LIN {X 0,Y 474.663,Z 446.241,A -85,B 0,C 180,E1 -7299.158,E2 -7299.158} C_VEL
LIN {X 0,Y 474.945,Z 438.322,A -85,B 0,C 180,E1 -7299.905,E2 -7299.905} C_VEL
LIN {X 0,Y 475.196,Z 429.952,A -85,B 0,C 180,E1 -7300.546,E2 -7300.546} C_VEL
LIN {X 0,Y 475.533,Z 419.253,A -85,B 0,C 180,E1 -7301.185,E2 -7301.185} C_VEL
LIN {X 0,Y 475.767,Z 407.58,A -85,B 0,C 180,E1 -7301.665,E2 -7301.665} C_VEL
LIN {X 0,Y 476.072,Z 397.775,A -85,B 0,C 180,E1 -7301.927,E2 -7301.927} C_VEL
LIN {X 0,Y 476.288,Z 334.559,A -85,B 0,C 180,E1 -7302.914,E2 -7302.914} C_VEL
LIN {X 0,Y 474.47,Z 320.647,A -85,B 0,C 180,E1 -7303.185,E2 -7303.185} C_VEL
LIN {X 0,Y 474.912,Z 304.767,A -85,B 0,C 180,E1 -7306.33,E2 -7306.33} C_VEL
LIN {X 0,Y 475.219,Z 291.489,A -85,B 0,C 180,E1 -7308.987,E2 -7308.987} C_VEL
LIN {X 0,Y 475.693,Z 278.163,A -85,B 0,C 180,E1 -7311.675,E2 -7311.675} C_VEL
LIN {X 0,Y 474.63,Z 271.177,A -85,B 0,C 180,E1 -7313.207,E2 -7313.207} C_VEL
LIN {X 0,Y 474.589,Z 271.182,A -85,B 0,C 180,E1 -7316.375,E2 -7316.375} C_VEL
LIN {X 0,Y 474.596,Z 271.18,A -85,B 0,C 180,E1 -7319.253,E2 -7319.253} C_VEL
LIN {X 0,Y 474.609,Z 271.177,A -85,B 0,C 180,E1 -7322.429,E2 -7322.429} C_VEL
LIN {X 0,Y 474.607,Z 271.177,A -85,B 0,C 180,E1 -7325.468,E2 -7325.468} C_VEL
LIN {X 0,Y 474.605,Z 271.178,A -85,B 0,C 180,E1 -7328.457,E2 -7328.457} C_VEL
LIN {X 0,Y 474.606,Z 271.176,A -85,B 0,C 180,E1 -7331.785,E2 -7331.785} C_VEL
LIN {X 0,Y 474.608,Z 271.181,A -85,B 0,C 180,E1 -7335.297,E2 -7335.297} C_VEL
LIN {X 0,Y 474.612,Z 271.173,A -85,B 0,C 180,E1 -7338.214,E2 -7338.214} C_VEL
LIN {X 0,Y 474.601,Z 271.181,A -85,B 0,C 180,E1 -7341.542,E2 -7341.542} C_VEL
LIN {X 0,Y 474.617,Z 271.172,A -85,B 0,C 180,E1 -7344.725,E2 -7344.725} C_VEL
LIN {X 0,Y 474.624,Z 271.175,A -85,B 0,C 180,E1 -7347.787,E2 -7347.787} C_VEL
LIN {X 0,Y 474.611,Z 271.172,A -85,B 0,C 180,E1 -7350.884,E2 -7350.884} C_VEL
LIN {X 0,Y 474.641,Z 271.168,A -85,B 0,C 180,E1 -7353.627,E2 -7353.627} C_VEL
LIN {X 0,Y 474.622,Z 271.171,A -85,B 0,C 180,E1 -7356.641,E2 -7356.641} C_VEL
LIN {X 0,Y 474.641,Z 271.173,A -85,B 0,C 180,E1 -7360.089,E2 -7360.089} C_VEL
LIN {X 0,Y 474.633,Z 271.17,A -85,B 0,C 180,E1 -7362.774,E2 -7362.774} C_VEL
LIN {X 0,Y 474.632,Z 271.167,A -85,B 0,C 180,E1 -7365.421,E2 -7365.421} C_VEL
LIN {X 0,Y 474.692,Z 271.165,A -85,B 0,C 180,E1 -7368.037,E2 -7368.037} C_VEL
LIN {X 0,Y 474.714,Z 271.156,A -85,B 0,C 180,E1 -7371.486,E2 -7371.486} C_VEL
LIN {X 0,Y 474.761,Z 271.154,A -85,B 0,C 180,E1 -7374.052,E2 -7374.052} C_VEL
LIN {X 0,Y 474.879,Z 271.138,A -85,B 0,C 180,E1 -7377.455,E2 -7377.455} C_VEL
LIN {X 0,Y 474.844,Z 271.15,A -85,B 0,C 180,E1 -7380.848,E2 -7380.848} C_VEL
LIN {X 0,Y 474.879,Z 271.137,A -85,B 0,C 180,E1 -7382.545,E2 -7382.545} C_VEL
LIN {X 0,Y 474.747,Z 271.155,A -85,B 0,C 180,E1 -7385.948,E2 -7385.948} C_VEL
LIN {X 0,Y 474.714,Z 271.157,A -85,B 0,C 180,E1 -7388.514,E2 -7388.514} C_VEL
LIN {X 0,Y 474.691,Z 271.161,A -85,B 0,C 180,E1 -7391.963,E2 -7391.963} C_VEL
LIN {X 0,Y 474.687,Z 271.172,A -85,B 0,C 180,E1 -7395.456,E2 -7395.456} C_VEL
LIN {X 0,Y 474.652,Z 271.171,A -85,B 0,C 180,E1 -7399.011,E2 -7399.011} C_VEL
LIN {X 0,Y 474.578,Z 271.186,A -85,B 0,C 180,E1 -7401.73,E2 -7401.73} C_VEL
LIN {X 0,Y 474.648,Z 271.171,A -85,B 0,C 180,E1 -7404.494,E2 -7404.494} C_VEL
LIN {X 0,Y 474.689,Z 271.165,A -85,B 0,C 180,E1 -7407.339,E2 -7407.339} C_VEL
LIN {X 0,Y 474.599,Z 271.175,A -85,B 0,C 180,E1 -7410.812,E2 -7410.812} C_VEL
LIN {X 0,Y 474.63,Z 271.178,A -85,B 0,C 180,E1 -7413.985,E2 -7413.985} C_VEL
LIN {X 0,Y 474.567,Z 271.181,A -85,B 0,C 180,E1 -7416.901,E2 -7416.901} C_VEL
LIN {X 0,Y 474.643,Z 271.172,A -85,B 0,C 180,E1 -7419.652,E2 -7419.652} C_VEL
LIN {X 0,Y 474.67,Z 271.173,A -85,B 0,C 180,E1 -7422.928,E2 -7422.928} C_VEL
LIN {X 0,Y 474.739,Z 271.319,A -85,B 0,C 180,E1 -7423.547,E2 -7423.547} C_VEL
LIN {X 0,Y 474.742,Z 280.743,A -85,B 0,C 180,E1 -7425.594,E2 -7425.594} C_VEL
LIN {X 0,Y 474.571,Z 295.866,A -85,B 0,C 180,E1 -7428.877,E2 -7428.877} C_VEL
LIN {X 0,Y 476.56,Z 308.996,A -85,B 0,C 180,E1 -7429.138,E2 -7429.138} C_VEL
LIN {X 0,Y 476.074,Z 372.113,A -85,B 0,C 180,E1 -7430.117,E2 -7430.117} C_VEL
LIN {X 0,Y 475.952,Z 381.875,A -85,B 0,C 180,E1 -7430.383,E2 -7430.383} C_VEL
LIN {X 0,Y 475.739,Z 393.015,A -85,B 0,C 180,E1 -7430.838,E2 -7430.838} C_VEL
LIN {X 0,Y 475.383,Z 404.114,A -85,B 0,C 180,E1 -7431.497,E2 -7431.497} C_VEL
LIN {X 0,Y 475.112,Z 412.388,A -85,B 0,C 180,E1 -7432.131,E2 -7432.131} C_VEL
LIN {X 0,Y 474.847,Z 419.279,A -85,B 0,C 180,E1 -7432.772,E2 -7432.772} C_VEL
LIN {X 0,Y 474.633,Z 425.51,A -85,B 0,C 180,E1 -7433.463,E2 -7433.463} C_VEL
LIN {X 0,Y 474.401,Z 432.473,A -85,B 0,C 180,E1 -7434.401,E2 -7434.401} C_VEL
LIN {X 0,Y 474.202,Z 437.454,A -85,B 0,C 180,E1 -7435.209,E2 -7435.209} C_VEL
LIN {X 0,Y 474.096,Z 442.083,A -85,B 0,C 180,E1 -7436.114,E2 -7436.114} C_VEL
LIN {X 0,Y 473.939,Z 445.242,A -85,B 0,C 180,E1 -7436.845,E2 -7436.845} C_VEL
LIN {X 0,Y 473.214,Z 447.665,A -85,B 0,C 180,E1 -7437.499,E2 -7437.499} C_VEL
LIN {X 0,Y 471.579,Z 449.734,A -85,B 0,C 180,E1 -7438.147,E2 -7438.147} C_VEL
LIN {X 0,Y 467.774,Z 452.844,A -85,B 0,C 180,E1 -7439.474,E2 -7439.474} C_VEL
LIN {X 0,Y 466.671,Z 453.932,A -85,B 0,C 180,E1 -7440.177,E2 -7440.177} C_VEL
LIN {X 0,Y 466.563,Z 454.183,A -85,B 0,C 180,E1 -7440.417,E2 -7440.417} C_VEL
LIN {X 0,Y 466.523,Z 454.848,A -85,B 0,C 180,E1 -7441.18,E2 -7441.18} C_VEL
LIN {X 0,Y 466.5,Z 455.117,A -85,B 0,C 180,E1 -7442.16,E2 -7442.16} C_VEL
LIN {X 0,Y 466.54,Z 454.729,A -85,B 0,C 180,E1 -7443.134,E2 -7443.134} C_VEL
LIN {X 0,Y 466.555,Z 453.682,A -85,B 0,C 180,E1 -7444.098,E2 -7444.098} C_VEL
LIN {X 0,Y 466.732,Z 450.926,A -85,B 0,C 180,E1 -7445.539,E2 -7445.539} C_VEL
LIN {X 0,Y 466.843,Z 447.631,A -85,B 0,C 180,E1 -7446.681,E2 -7446.681} C_VEL
LIN {X 0,Y 466.947,Z 443.943,A -85,B 0,C 180,E1 -7447.665,E2 -7447.665} C_VEL
LIN {X 0,Y 467.086,Z 439.593,A -85,B 0,C 180,E1 -7448.601,E2 -7448.601} C_VEL
LIN {X 0,Y 467.295,Z 434.283,A -85,B 0,C 180,E1 -7449.533,E2 -7449.533} C_VEL
LIN {X 0,Y 467.54,Z 427.826,A -85,B 0,C 180,E1 -7450.461,E2 -7450.461} C_VEL
LIN {X 0,Y 467.766,Z 421.819,A -85,B 0,C 180,E1 -7451.183,E2 -7451.183} C_VEL
LIN {X 0,Y 468.079,Z 413.97,A -85,B 0,C 180,E1 -7451.961,E2 -7451.961} C_VEL
LIN {X 0,Y 468.322,Z 406.975,A -85,B 0,C 180,E1 -7452.535,E2 -7452.535} C_VEL
LIN {X 0,Y 468.602,Z 398.339,A -85,B 0,C 180,E1 -7453.108,E2 -7453.108} C_VEL
LIN {X 0,Y 468.824,Z 390.258,A -85,B 0,C 180,E1 -7453.531,E2 -7453.531} C_VEL
LIN {X 0,Y 468.982,Z 381.301,A -85,B 0,C 180,E1 -7453.885,E2 -7453.885} C_VEL
LIN {X 0,Y 469.169,Z 371.936,A -85,B 0,C 180,E1 -7454.137,E2 -7454.137} C_VEL
LIN {X 0,Y 469.47,Z 308.099,A -85,B 0,C 180,E1 -7455.146,E2 -7455.146} C_VEL
LIN {X 0,Y 467.529,Z 296.318,A -85,B 0,C 180,E1 -7455.389,E2 -7455.389} C_VEL
LIN {X 0,Y 467.842,Z 284.205,A -85,B 0,C 180,E1 -7458.3,E2 -7458.3} C_VEL
LIN {X 0,Y 467.997,Z 275.173,A -85,B 0,C 180,E1 -7460.492,E2 -7460.492} C_VEL
LIN {X 0,Y 467.731,Z 272.039,A -85,B 0,C 180,E1 -7461.304,E2 -7461.304} C_VEL
LIN {X 0,Y 467.736,Z 272.036,A -85,B 0,C 180,E1 -7463.963,E2 -7463.963} C_VEL
LIN {X 0,Y 467.86,Z 272.017,A -85,B 0,C 180,E1 -7467.417,E2 -7467.417} C_VEL
LIN {X 0,Y 467.884,Z 272.018,A -85,B 0,C 180,E1 -7470,E2 -7470} C_VEL
LIN {X 0,Y 467.861,Z 272.015,A -85,B 0,C 180,E1 -7472.583,E2 -7472.583} C_VEL
LIN {X 0,Y 467.722,Z 272.038,A -85,B 0,C 180,E1 -7476.037,E2 -7476.037} C_VEL
LIN {X 0,Y 467.682,Z 272.039,A -85,B 0,C 180,E1 -7478.642,E2 -7478.642} C_VEL
LIN {X 0,Y 467.657,Z 272.045,A -85,B 0,C 180,E1 -7482.145,E2 -7482.145} C_VEL
LIN {X 0,Y 467.64,Z 272.041,A -85,B 0,C 180,E1 -7485.694,E2 -7485.694} C_VEL
LIN {X 0,Y 467.613,Z 272.05,A -85,B 0,C 180,E1 -7488.762,E2 -7488.762} C_VEL
LIN {X 0,Y 467.58,Z 272.05,A -85,B 0,C 180,E1 -7491.267,E2 -7491.267} C_VEL
LIN {X 0,Y 467.57,Z 272.05,A -85,B 0,C 180,E1 -7493.943,E2 -7493.943} C_VEL
LIN {X 0,Y 467.615,Z 272.052,A -85,B 0,C 180,E1 -7496.8,E2 -7496.8} C_VEL
LIN {X 0,Y 467.552,Z 272.052,A -85,B 0,C 180,E1 -7499.737,E2 -7499.737} C_VEL
LIN {X 0,Y 467.576,Z 272.053,A -85,B 0,C 180,E1 -7502.758,E2 -7502.758} C_VEL
LIN {X 0,Y 467.549,Z 272.053,A -85,B 0,C 180,E1 -7505.889,E2 -7505.889} C_VEL
LIN {X 0,Y 467.577,Z 272.055,A -85,B 0,C 180,E1 -7509.144,E2 -7509.144} C_VEL
LIN {X 0,Y 467.581,Z 272.048,A -85,B 0,C 180,E1 -7512.566,E2 -7512.566} C_VEL
LIN {X 0,Y 467.564,Z 272.053,A -85,B 0,C 180,E1 -7515.052,E2 -7515.052} C_VEL
LIN {X 0,Y 467.618,Z 272.05,A -85,B 0,C 180,E1 -7517.443,E2 -7517.443} C_VEL
LIN {X 0,Y 467.592,Z 272.047,A -85,B 0,C 180,E1 -7520.856,E2 -7520.856} C_VEL
LIN {X 0,Y 467.555,Z 272.054,A -85,B 0,C 180,E1 -7524.259,E2 -7524.259} C_VEL
LIN {X 0,Y 467.573,Z 272.05,A -85,B 0,C 180,E1 -7527.32,E2 -7527.32} C_VEL
LIN {X 0,Y 467.568,Z 272.051,A -85,B 0,C 180,E1 -7530.665,E2 -7530.665} C_VEL
LIN {X 0,Y 467.617,Z 272.043,A -85,B 0,C 180,E1 -7533.2,E2 -7533.2} C_VEL
LIN {X 0,Y 467.582,Z 272.054,A -85,B 0,C 180,E1 -7536.467,E2 -7536.467} C_VEL
LIN {X 0,Y 467.611,Z 272.046,A -85,B 0,C 180,E1 -7539.777,E2 -7539.777} C_VEL
LIN {X 0,Y 467.597,Z 272.055,A -85,B 0,C 180,E1 -7542.506,E2 -7542.506} C_VEL
LIN {X 0,Y 467.593,Z 272.048,A -85,B 0,C 180,E1 -7545.196,E2 -7545.196} C_VEL
LIN {X 0,Y 467.643,Z 272.041,A -85,B 0,C 180,E1 -7547.854,E2 -7547.854} C_VEL
LIN {X 0,Y 467.669,Z 272.039,A -85,B 0,C 180,E1 -7551.357,E2 -7551.357} C_VEL
LIN {X 0,Y 467.722,Z 272.03,A -85,B 0,C 180,E1 -7553.962,E2 -7553.962} C_VEL
LIN {X 0,Y 467.846,Z 272.018,A -85,B 0,C 180,E1 -7557.417,E2 -7557.417} C_VEL
LIN {X 0,Y 467.867,Z 272.012,A -85,B 0,C 180,E1 -7560,E2 -7560} C_VEL
LIN {X 0,Y 467.846,Z 272.016,A -85,B 0,C 180,E1 -7562.583,E2 -7562.583} C_VEL
LIN {X 0,Y 467.725,Z 272.031,A -85,B 0,C 180,E1 -7566.038,E2 -7566.038} C_VEL
LIN {X 0,Y 467.669,Z 272.037,A -85,B 0,C 180,E1 -7568.643,E2 -7568.643} C_VEL
LIN {X 0,Y 467.671,Z 272.038,A -85,B 0,C 180,E1 -7572.145,E2 -7572.145} C_VEL
LIN {X 0,Y 467.637,Z 272.047,A -85,B 0,C 180,E1 -7575.885,E2 -7575.885} C_VEL
LIN {X 0,Y 467.611,Z 272.047,A -85,B 0,C 180,E1 -7579.308,E2 -7579.308} C_VEL
LIN {X 0,Y 467.523,Z 272.061,A -85,B 0,C 180,E1 -7582.074,E2 -7582.074} C_VEL
LIN {X 0,Y 467.592,Z 272.047,A -85,B 0,C 180,E1 -7584.888,E2 -7584.888} C_VEL
LIN {X 0,Y 467.608,Z 272.049,A -85,B 0,C 180,E1 -7587.77,E2 -7587.77} C_VEL
LIN {X 0,Y 467.557,Z 272.051,A -85,B 0,C 180,E1 -7591.045,E2 -7591.045} C_VEL
LIN {X 0,Y 467.58,Z 272.056,A -85,B 0,C 180,E1 -7594.243,E2 -7594.243} C_VEL
LIN {X 0,Y 467.539,Z 272.054,A -85,B 0,C 180,E1 -7597.187,E2 -7597.187} C_VEL
LIN {X 0,Y 467.566,Z 272.055,A -85,B 0,C 180,E1 -7600.266,E2 -7600.266} C_VEL
LIN {X 0,Y 467.579,Z 272.057,A -85,B 0,C 180,E1 -7602.568,E2 -7602.568} C_VEL
LIN {X 0,Y 467.558,Z 272.055,A -85,B 0,C 180,E1 -7605.053,E2 -7605.053} C_VEL
LIN {X 0,Y 467.565,Z 272.056,A -85,B 0,C 180,E1 -7608.597,E2 -7608.597} C_VEL
LIN {X 0,Y 467.559,Z 272.051,A -85,B 0,C 180,E1 -7611.956,E2 -7611.956} C_VEL
LIN {X 0,Y 467.553,Z 272.059,A -85,B 0,C 180,E1 -7615.168,E2 -7615.168} C_VEL
LIN {X 0,Y 467.577,Z 272.048,A -85,B 0,C 180,E1 -7618.261,E2 -7618.261} C_VEL
LIN {X 0,Y 467.551,Z 272.061,A -85,B 0,C 180,E1 -7621.25,E2 -7621.25} C_VEL
LIN {X 0,Y 467.565,Z 272.053,A -85,B 0,C 180,E1 -7624.158,E2 -7624.158} C_VEL
LIN {X 0,Y 467.609,Z 272.073,A -85,B 0,C 180,E1 -7626.464,E2 -7626.464} C_VEL
LIN {X 0,Y 468.776,Z 278.945,A -85,B 0,C 180,E1 -7627.988,E2 -7627.988} C_VEL
LIN {X 0,Y 468.56,Z 287.645,A -85,B 0,C 180,E1 -7629.82,E2 -7629.82} C_VEL
LIN {X 0,Y 468.008,Z 303.938,A -85,B 0,C 180,E1 -7633.198,E2 -7633.198} C_VEL
LIN {X 0,Y 467.474,Z 320.66,A -85,B 0,C 180,E1 -7636.619,E2 -7636.619} C_VEL
LIN {X 0,Y 469.474,Z 337.921,A -85,B 0,C 180,E1 -7636.966,E2 -7636.966} C_VEL
LIN {X 0,Y 469.076,Z 398.227,A -85,B 0,C 180,E1 -7637.92,E2 -7637.92} C_VEL
LIN {X 0,Y 468.802,Z 408.676,A -85,B 0,C 180,E1 -7638.214,E2 -7638.214} C_VEL
LIN {X 0,Y 468.482,Z 420.839,A -85,B 0,C 180,E1 -7638.754,E2 -7638.754} C_VEL
LIN {X 0,Y 468.211,Z 429.659,A -85,B 0,C 180,E1 -7639.295,E2 -7639.295} C_VEL
LIN {X 0,Y 467.919,Z 438.06,A -85,B 0,C 180,E1 -7639.945,E2 -7639.945} C_VEL
LIN {X 0,Y 467.619,Z 445.999,A -85,B 0,C 180,E1 -7640.703,E2 -7640.703} C_VEL
LIN {X 0,Y 467.305,Z 453.415,A -85,B 0,C 180,E1 -7641.568,E2 -7641.568} C_VEL
LIN {X 0,Y 467.048,Z 460.937,A -85,B 0,C 180,E1 -7642.652,E2 -7642.652} C_VEL
LIN {X 0,Y 466.87,Z 467.813,A -85,B 0,C 180,E1 -7643.951,E2 -7643.951} C_VEL
LIN {X 0,Y 466.72,Z 473.018,A -85,B 0,C 180,E1 -7645.249,E2 -7645.249} C_VEL
LIN {X 0,Y 466.706,Z 475.684,A -85,B 0,C 180,E1 -7646.115,E2 -7646.115} C_VEL
LIN {X 0,Y 466.666,Z 478.604,A -85,B 0,C 180,E1 -7647.411,E2 -7647.411} C_VEL
LIN {X 0,Y 466.606,Z 479.865,A -85,B 0,C 180,E1 -7648.274,E2 -7648.274} C_VEL
LIN {X 0,Y 466.616,Z 480.652,A -85,B 0,C 180,E1 -7649.137,E2 -7649.137} C_VEL
LIN {X 0,Y 466.597,Z 480.945,A -85,B 0,C 180,E1 -7650,E2 -7650} C_VEL
LIN {X 0,Y 466.616,Z 480.646,A -85,B 0,C 180,E1 -7650.863,E2 -7650.863} C_VEL
LIN {X 0,Y 466.606,Z 479.86,A -85,B 0,C 180,E1 -7651.726,E2 -7651.726} C_VEL
LIN {X 0,Y 466.666,Z 478.599,A -85,B 0,C 180,E1 -7652.589,E2 -7652.589} C_VEL
LIN {X 0,Y 466.706,Z 475.676,A -85,B 0,C 180,E1 -7653.885,E2 -7653.885} C_VEL
LIN {X 0,Y 466.72,Z 473.012,A -85,B 0,C 180,E1 -7654.751,E2 -7654.751} C_VEL
LIN {X 0,Y 466.857,Z 467.805,A -85,B 0,C 180,E1 -7656.049,E2 -7656.049} C_VEL
LIN {X 0,Y 467.048,Z 460.944,A -85,B 0,C 180,E1 -7657.348,E2 -7657.348} C_VEL
LIN {X 0,Y 467.305,Z 453.449,A -85,B 0,C 180,E1 -7658.432,E2 -7658.432} C_VEL
LIN {X 0,Y 467.62,Z 446.06,A -85,B 0,C 180,E1 -7659.297,E2 -7659.297} C_VEL
LIN {X 0,Y 467.938,Z 438.149,A -85,B 0,C 180,E1 -7660.055,E2 -7660.055} C_VEL
LIN {X 0,Y 468.216,Z 429.79,A -85,B 0,C 180,E1 -7660.705,E2 -7660.705} C_VEL
LIN {X 0,Y 468.567,Z 419.109,A -85,B 0,C 180,E1 -7661.353,E2 -7661.353} C_VEL
LIN {X 0,Y 468.837,Z 407.471,A -85,B 0,C 180,E1 -7661.84,E2 -7661.84} C_VEL
LIN {X 0,Y 469.142,Z 397.719,A -85,B 0,C 180,E1 -7662.106,E2 -7662.106} C_VEL
LIN {X 0,Y 469.384,Z 335.49,A -85,B 0,C 180,E1 -7663.093,E2 -7663.093} C_VEL
LIN {X 0,Y 467.442,Z 320.385,A -85,B 0,C 180,E1 -7663.399,E2 -7663.399} C_VEL
LIN {X 0,Y 467.903,Z 304.556,A -85,B 0,C 180,E1 -7666.581,E2 -7666.581} C_VEL
LIN {X 0,Y 468.219,Z 292.753,A -85,B 0,C 180,E1 -7668.98,E2 -7668.98} C_VEL
LIN {X 0,Y 468.703,Z 279.867,A -85,B 0,C 180,E1 -7671.618,E2 -7671.618} C_VEL
LIN {X 0,Y 467.897,Z 273.478,A -85,B 0,C 180,E1 -7672.987,E2 -7672.987} C_VEL
LIN {X 0,Y 467.6,Z 272.053,A -85,B 0,C 180,E1 -7673.315,E2 -7673.315} C_VEL
LIN {X 0,Y 467.564,Z 272.055,A -85,B 0,C 180,E1 -7675.842,E2 -7675.842} C_VEL
LIN {X 0,Y 467.541,Z 272.061,A -85,B 0,C 180,E1 -7678.751,E2 -7678.751} C_VEL
LIN {X 0,Y 467.576,Z 272.05,A -85,B 0,C 180,E1 -7681.739,E2 -7681.739} C_VEL
LIN {X 0,Y 467.553,Z 272.06,A -85,B 0,C 180,E1 -7684.832,E2 -7684.832} C_VEL
LIN {X 0,Y 467.558,Z 272.055,A -85,B 0,C 180,E1 -7688.044,E2 -7688.044} C_VEL
LIN {X 0,Y 467.565,Z 272.057,A -85,B 0,C 180,E1 -7691.403,E2 -7691.403} C_VEL
LIN {X 0,Y 467.558,Z 272.059,A -85,B 0,C 180,E1 -7695.052,E2 -7695.052} C_VEL
LIN {X 0,Y 467.581,Z 272.057,A -85,B 0,C 180,E1 -7697.439,E2 -7697.439} C_VEL
LIN {X 0,Y 467.55,Z 272.054,A -85,B 0,C 180,E1 -7700.852,E2 -7700.852} C_VEL
LIN {X 0,Y 467.552,Z 272.054,A -85,B 0,C 180,E1 -7704.26,E2 -7704.26} C_VEL
LIN {X 0,Y 467.571,Z 272.05,A -85,B 0,C 180,E1 -7707.32,E2 -7707.32} C_VEL
LIN {X 0,Y 467.557,Z 272.051,A -85,B 0,C 180,E1 -7710.667,E2 -7710.667} C_VEL
LIN {X 0,Y 467.601,Z 272.041,A -85,B 0,C 180,E1 -7713.199,E2 -7713.199} C_VEL
LIN {X 0,Y 467.578,Z 272.05,A -85,B 0,C 180,E1 -7716.468,E2 -7716.468} C_VEL
LIN {X 0,Y 467.609,Z 272.044,A -85,B 0,C 180,E1 -7719.777,E2 -7719.777} C_VEL
LIN {X 0,Y 467.592,Z 272.05,A -85,B 0,C 180,E1 -7722.506,E2 -7722.506} C_VEL
LIN {X 0,Y 467.59,Z 272.044,A -85,B 0,C 180,E1 -7725.196,E2 -7725.196} C_VEL
LIN {X 0,Y 467.644,Z 272.042,A -85,B 0,C 180,E1 -7727.854,E2 -7727.854} C_VEL
LIN {X 0,Y 467.668,Z 272.034,A -85,B 0,C 180,E1 -7731.357,E2 -7731.357} C_VEL
LIN {X 0,Y 467.724,Z 272.03,A -85,B 0,C 180,E1 -7733.962,E2 -7733.962} C_VEL
LIN {X 0,Y 467.845,Z 272.014,A -85,B 0,C 180,E1 -7737.417,E2 -7737.417} C_VEL
LIN {X 0,Y 467.866,Z 272.012,A -85,B 0,C 180,E1 -7740,E2 -7740} C_VEL
LIN {X 0,Y 467.845,Z 272.013,A -85,B 0,C 180,E1 -7742.583,E2 -7742.583} C_VEL
LIN {X 0,Y 467.709,Z 272.032,A -85,B 0,C 180,E1 -7746.038,E2 -7746.038} C_VEL
LIN {X 0,Y 467.668,Z 272.036,A -85,B 0,C 180,E1 -7748.643,E2 -7748.643} C_VEL
LIN {X 0,Y 467.643,Z 272.037,A -85,B 0,C 180,E1 -7752.146,E2 -7752.146} C_VEL
LIN {X 0,Y 467.626,Z 272.047,A -85,B 0,C 180,E1 -7755.696,E2 -7755.696} C_VEL
LIN {X 0,Y 467.605,Z 272.048,A -85,B 0,C 180,E1 -7758.765,E2 -7758.765} C_VEL
LIN {X 0,Y 467.569,Z 272.053,A -85,B 0,C 180,E1 -7761.269,E2 -7761.269} C_VEL
LIN {X 0,Y 467.562,Z 272.058,A -85,B 0,C 180,E1 -7763.944,E2 -7763.944} C_VEL
LIN {X 0,Y 467.617,Z 272.044,A -85,B 0,C 180,E1 -7766.8,E2 -7766.8} C_VEL
LIN {X 0,Y 467.576,Z 272.054,A -85,B 0,C 180,E1 -7769.737,E2 -7769.737} C_VEL
LIN {X 0,Y 467.574,Z 272.052,A -85,B 0,C 180,E1 -7772.759,E2 -7772.759} C_VEL
LIN {X 0,Y 467.548,Z 272.056,A -85,B 0,C 180,E1 -7775.89,E2 -7775.89} C_VEL
LIN {X 0,Y 467.592,Z 272.05,A -85,B 0,C 180,E1 -7779.144,E2 -7779.144} C_VEL
LIN {X 0,Y 467.613,Z 272.053,A -85,B 0,C 180,E1 -7782.572,E2 -7782.572} C_VEL
LIN {X 0,Y 467.692,Z 272.169,A -85,B 0,C 180,E1 -7783.431,E2 -7783.431} C_VEL
LIN {X 0,Y 467.757,Z 280.981,A -85,B 0,C 180,E1 -7785.372,E2 -7785.372} C_VEL
LIN {X 0,Y 467.529,Z 295.966,A -85,B 0,C 180,E1 -7788.662,E2 -7788.662} C_VEL
LIN {X 0,Y 469.614,Z 308.501,A -85,B 0,C 180,E1 -7788.928,E2 -7788.928} C_VEL
LIN {X 0,Y 469.139,Z 372.245,A -85,B 0,C 180,E1 -7789.933,E2 -7789.933} C_VEL
LIN {X 0,Y 469.024,Z 381.964,A -85,B 0,C 180,E1 -7790.201,E2 -7790.201} C_VEL
LIN {X 0,Y 468.818,Z 392.478,A -85,B 0,C 180,E1 -7790.633,E2 -7790.633} C_VEL
LIN {X 0,Y 468.438,Z 403.494,A -85,B 0,C 180,E1 -7791.275,E2 -7791.275} C_VEL
LIN {X 0,Y 468.105,Z 412.934,A -85,B 0,C 180,E1 -7792.009,E2 -7792.009} C_VEL
LIN {X 0,Y 467.803,Z 420.829,A -85,B 0,C 180,E1 -7792.773,E2 -7792.773} C_VEL
LIN {X 0,Y 467.546,Z 427.649,A -85,B 0,C 180,E1 -7793.578,E2 -7793.578} C_VEL
LIN {X 0,Y 467.287,Z 434.861,A -85,B 0,C 180,E1 -7794.618,E2 -7794.618} C_VEL
LIN {X 0,Y 467.046,Z 441.555,A -85,B 0,C 180,E1 -7795.856,E2 -7795.856} C_VEL
LIN {X 0,Y 466.865,Z 445.626,A -85,B 0,C 180,E1 -7796.813,E2 -7796.813} C_VEL
LIN {X 0,Y 466.76,Z 450.059,A -85,B 0,C 180,E1 -7798.199,E2 -7798.199} C_VEL
LIN {X 0,Y 466.667,Z 452.364,A -85,B 0,C 180,E1 -7799.201,E2 -7799.201} C_VEL
LIN {X 0,Y 466.563,Z 454.183,A -85,B 0,C 180,E1 -7800.417,E2 -7800.417} C_VEL
LIN {X 0,Y 465.835,Z 454.858,A -85,B 0,C 180,E1 -7801.133,E2 -7801.133} C_VEL
LIN {X 0,Y 462.926,Z 455.162,A -85,B 0,C 180,E1 -7802.302,E2 -7802.302} C_VEL
LIN {X 0,Y 460.075,Z 454.587,A -85,B 0,C 180,E1 -7803.484,E2 -7803.484} C_VEL
LIN {X 0,Y 459.453,Z 453.679,A -85,B 0,C 180,E1 -7804.213,E2 -7804.213} C_VEL
LIN {X 0,Y 459.653,Z 451.038,A -85,B 0,C 180,E1 -7805.618,E2 -7805.618} C_VEL
LIN {X 0,Y 459.744,Z 448.396,A -85,B 0,C 180,E1 -7806.582,E2 -7806.582} C_VEL
LIN {X 0,Y 459.878,Z 444.004,A -85,B 0,C 180,E1 -7807.776,E2 -7807.776} C_VEL
LIN {X 0,Y 460.026,Z 439.568,A -85,B 0,C 180,E1 -7808.737,E2 -7808.737} C_VEL
LIN {X 0,Y 460.25,Z 434.28,A -85,B 0,C 180,E1 -7809.673,E2 -7809.673} C_VEL
LIN {X 0,Y 460.521,Z 428.073,A -85,B 0,C 180,E1 -7810.577,E2 -7810.577} C_VEL
LIN {X 0,Y 460.798,Z 420.905,A -85,B 0,C 180,E1 -7811.436,E2 -7811.436} C_VEL
LIN {X 0,Y 461.111,Z 413.802,A -85,B 0,C 180,E1 -7812.138,E2 -7812.138} C_VEL
LIN {X 0,Y 461.371,Z 406.725,A -85,B 0,C 180,E1 -7812.721,E2 -7812.721} C_VEL
LIN {X 0,Y 461.634,Z 398.122,A -85,B 0,C 180,E1 -7813.294,E2 -7813.294} C_VEL
LIN {X 0,Y 461.867,Z 390.139,A -85,B 0,C 180,E1 -7813.713,E2 -7813.713} C_VEL
LIN {X 0,Y 462.045,Z 380.541,A -85,B 0,C 180,E1 -7814.091,E2 -7814.091} C_VEL
LIN {X 0,Y 462.232,Z 370.811,A -85,B 0,C 180,E1 -7814.343,E2 -7814.343} C_VEL
LIN {X 0,Y 462.478,Z 308.494,A -85,B 0,C 180,E1 -7815.339,E2 -7815.339} C_VEL
LIN {X 0,Y 460.484,Z 296.423,A -85,B 0,C 180,E1 -7815.612,E2 -7815.612} C_VEL
LIN {X 0,Y 460.831,Z 284.28,A -85,B 0,C 180,E1 -7818.565,E2 -7818.565} C_VEL
LIN {X 0,Y 460.928,Z 275.249,A -85,B 0,C 180,E1 -7820.788,E2 -7820.788} C_VEL
LIN {X 0,Y 460.722,Z 272.912,A -85,B 0,C 180,E1 -7821.392,E2 -7821.392} C_VEL
LIN {X 0,Y 460.695,Z 272.906,A -85,B 0,C 180,E1 -7824.748,E2 -7824.748} C_VEL
LIN {X 0,Y 460.801,Z 272.895,A -85,B 0,C 180,E1 -7827.378,E2 -7827.378} C_VEL
LIN {X 0,Y 460.855,Z 272.894,A -85,B 0,C 180,E1 -7830,E2 -7830} C_VEL
LIN {X 0,Y 460.802,Z 272.894,A -85,B 0,C 180,E1 -7832.622,E2 -7832.622} C_VEL
LIN {X 0,Y 460.686,Z 272.916,A -85,B 0,C 180,E1 -7836.13,E2 -7836.13} C_VEL
LIN {X 0,Y 460.629,Z 272.916,A -85,B 0,C 180,E1 -7838.776,E2 -7838.776} C_VEL
LIN {X 0,Y 460.615,Z 272.924,A -85,B 0,C 180,E1 -7842.444,E2 -7842.444} C_VEL
LIN {X 0,Y 460.601,Z 272.92,A -85,B 0,C 180,E1 -7845.997,E2 -7845.997} C_VEL
LIN {X 0,Y 460.568,Z 272.922,A -85,B 0,C 180,E1 -7849.615,E2 -7849.615} C_VEL
LIN {X 0,Y 460.511,Z 272.934,A -85,B 0,C 180,E1 -7852.428,E2 -7852.428} C_VEL
LIN {X 0,Y 460.556,Z 272.923,A -85,B 0,C 180,E1 -7855.798,E2 -7855.798} C_VEL
LIN {X 0,Y 460.551,Z 272.925,A -85,B 0,C 180,E1 -7858.232,E2 -7858.232} C_VEL
LIN {X 0,Y 460.518,Z 272.933,A -85,B 0,C 180,E1 -7861.282,E2 -7861.282} C_VEL
LIN {X 0,Y 460.519,Z 272.929,A -85,B 0,C 180,E1 -7864.503,E2 -7864.503} C_VEL
LIN {X 0,Y 460.497,Z 272.934,A -85,B 0,C 180,E1 -7867.622,E2 -7867.622} C_VEL
LIN {X 0,Y 460.537,Z 272.926,A -85,B 0,C 180,E1 -7870.268,E2 -7870.268} C_VEL
LIN {X 0,Y 460.495,Z 272.939,A -85,B 0,C 180,E1 -7873.374,E2 -7873.374} C_VEL
LIN {X 0,Y 460.518,Z 272.928,A -85,B 0,C 180,E1 -7876.627,E2 -7876.627} C_VEL
LIN {X 0,Y 460.552,Z 272.932,A -85,B 0,C 180,E1 -7879.727,E2 -7879.727} C_VEL
LIN {X 0,Y 460.52,Z 272.928,A -85,B 0,C 180,E1 -7882.518,E2 -7882.518} C_VEL
LIN {X 0,Y 460.54,Z 272.93,A -85,B 0,C 180,E1 -7885.623,E2 -7885.623} C_VEL
LIN {X 0,Y 460.528,Z 272.927,A -85,B 0,C 180,E1 -7888.744,E2 -7888.744} C_VEL
LIN {X 0,Y 460.549,Z 272.928,A -85,B 0,C 180,E1 -7891.767,E2 -7891.767} C_VEL
LIN {X 0,Y 460.549,Z 272.926,A -85,B 0,C 180,E1 -7894.705,E2 -7894.705} C_VEL
LIN {X 0,Y 460.5,Z 272.931,A -85,B 0,C 180,E1 -7897.571,E2 -7897.571} C_VEL
LIN {X 0,Y 460.557,Z 272.932,A -85,B 0,C 180,E1 -7900.384,E2 -7900.384} C_VEL
LIN {X 0,Y 460.553,Z 272.925,A -85,B 0,C 180,E1 -7903.146,E2 -7903.146} C_VEL
LIN {X 0,Y 460.545,Z 272.925,A -85,B 0,C 180,E1 -7905.868,E2 -7905.868} C_VEL
LIN {X 0,Y 460.598,Z 272.925,A -85,B 0,C 180,E1 -7908.559,E2 -7908.559} C_VEL
LIN {X 0,Y 460.682,Z 272.908,A -85,B 0,C 180,E1 -7912.108,E2 -7912.108} C_VEL
LIN {X 0,Y 460.681,Z 272.914,A -85,B 0,C 180,E1 -7914.748,E2 -7914.748} C_VEL
LIN {X 0,Y 460.811,Z 272.895,A -85,B 0,C 180,E1 -7917.377,E2 -7917.377} C_VEL
LIN {X 0,Y 460.838,Z 272.888,A -85,B 0,C 180,E1 -7920,E2 -7920} C_VEL
LIN {X 0,Y 460.787,Z 272.896,A -85,B 0,C 180,E1 -7922.622,E2 -7922.622} C_VEL
LIN {X 0,Y 460.691,Z 272.907,A -85,B 0,C 180,E1 -7926.13,E2 -7926.13} C_VEL
LIN {X 0,Y 460.616,Z 272.917,A -85,B 0,C 180,E1 -7928.776,E2 -7928.776} C_VEL
LIN {X 0,Y 460.622,Z 272.915,A -85,B 0,C 180,E1 -7932.457,E2 -7932.457} C_VEL
LIN {X 0,Y 460.588,Z 272.923,A -85,B 0,C 180,E1 -7935.998,E2 -7935.998} C_VEL
LIN {X 0,Y 460.558,Z 272.923,A -85,B 0,C 180,E1 -7938.902,E2 -7938.902} C_VEL
LIN {X 0,Y 460.504,Z 272.933,A -85,B 0,C 180,E1 -7941.486,E2 -7941.486} C_VEL
LIN {X 0,Y 460.531,Z 272.93,A -85,B 0,C 180,E1 -7944.333,E2 -7944.333} C_VEL
LIN {X 0,Y 460.561,Z 272.923,A -85,B 0,C 180,E1 -7947.244,E2 -7947.244} C_VEL
LIN {X 0,Y 460.499,Z 272.938,A -85,B 0,C 180,E1 -7950.241,E2 -7950.241} C_VEL
LIN {X 0,Y 460.519,Z 272.928,A -85,B 0,C 180,E1 -7953.326,E2 -7953.326} C_VEL
LIN {X 0,Y 460.468,Z 272.941,A -85,B 0,C 180,E1 -7956.53,E2 -7956.53} C_VEL
LIN {X 0,Y 460.516,Z 272.929,A -85,B 0,C 180,E1 -7959.864,E2 -7959.864} C_VEL
LIN {X 0,Y 460.505,Z 272.934,A -85,B 0,C 180,E1 -7962.901,E2 -7962.901} C_VEL
LIN {X 0,Y 460.498,Z 272.93,A -85,B 0,C 180,E1 -7965.832,E2 -7965.832} C_VEL
LIN {X 0,Y 460.52,Z 272.934,A -85,B 0,C 180,E1 -7968.989,E2 -7968.989} C_VEL
LIN {X 0,Y 460.515,Z 272.932,A -85,B 0,C 180,E1 -7971.267,E2 -7971.267} C_VEL
LIN {X 0,Y 460.503,Z 272.932,A -85,B 0,C 180,E1 -7974.555,E2 -7974.555} C_VEL
LIN {X 0,Y 460.525,Z 272.929,A -85,B 0,C 180,E1 -7977.716,E2 -7977.716} C_VEL
LIN {X 0,Y 460.522,Z 272.93,A -85,B 0,C 180,E1 -7980.769,E2 -7980.769} C_VEL
LIN {X 0,Y 460.516,Z 272.934,A -85,B 0,C 180,E1 -7983.733,E2 -7983.733} C_VEL
LIN {X 0,Y 460.581,Z 273.028,A -85,B 0,C 180,E1 -7986.336,E2 -7986.336} C_VEL
LIN {X 0,Y 461.848,Z 281.163,A -85,B 0,C 180,E1 -7988.162,E2 -7988.162} C_VEL
LIN {X 0,Y 461.425,Z 291.788,A -85,B 0,C 180,E1 -7990.423,E2 -7990.423} C_VEL
LIN {X 0,Y 460.838,Z 308.349,A -85,B 0,C 180,E1 -7993.9,E2 -7993.9} C_VEL
LIN {X 0,Y 460.416,Z 320.573,A -85,B 0,C 180,E1 -7996.435,E2 -7996.435} C_VEL
LIN {X 0,Y 462.542,Z 337.9,A -85,B 0,C 180,E1 -7996.776,E2 -7996.776} C_VEL
LIN {X 0,Y 462.148,Z 397.722,A -85,B 0,C 180,E1 -7997.736,E2 -7997.736} C_VEL
LIN {X 0,Y 461.878,Z 407.449,A -85,B 0,C 180,E1 -7998.007,E2 -7998.007} C_VEL
LIN {X 0,Y 461.609,Z 418.533,A -85,B 0,C 180,E1 -7998.473,E2 -7998.473} C_VEL
LIN {X 0,Y 461.207,Z 429.372,A -85,B 0,C 180,E1 -7999.131,E2 -7999.131} C_VEL
LIN {X 0,Y 460.919,Z 437.791,A -85,B 0,C 180,E1 -7999.79,E2 -7999.79} C_VEL
LIN {X 0,Y 460.575,Z 445.742,A -85,B 0,C 180,E1 -8000.559,E2 -8000.559} C_VEL
LIN {X 0,Y 460.259,Z 453.168,A -85,B 0,C 180,E1 -8001.438,E2 -8001.438} C_VEL
LIN {X 0,Y 459.977,Z 460.701,A -85,B 0,C 180,E1 -8002.538,E2 -8002.538} C_VEL
LIN {X 0,Y 459.781,Z 467.592,A -85,B 0,C 180,E1 -8003.858,E2 -8003.858} C_VEL
LIN {X 0,Y 459.651,Z 472.804,A -85,B 0,C 180,E1 -8005.176,E2 -8005.176} C_VEL
LIN {X 0,Y 459.6,Z 475.475,A -85,B 0,C 180,E1 -8006.054,E2 -8006.054} C_VEL
LIN {X 0,Y 459.59,Z 478.4,A -85,B 0,C 180,E1 -8007.371,E2 -8007.371} C_VEL
LIN {X 0,Y 459.519,Z 479.665,A -85,B 0,C 180,E1 -8008.247,E2 -8008.247} C_VEL
LIN {X 0,Y 459.519,Z 480.454,A -85,B 0,C 180,E1 -8009.124,E2 -8009.124} C_VEL
LIN {X 0,Y 459.529,Z 480.749,A -85,B 0,C 180,E1 -8010,E2 -8010} C_VEL
LIN {X 0,Y 459.519,Z 480.451,A -85,B 0,C 180,E1 -8010.876,E2 -8010.876} C_VEL
LIN {X 0,Y 459.519,Z 479.667,A -85,B 0,C 180,E1 -8011.753,E2 -8011.753} C_VEL
LIN {X 0,Y 459.59,Z 478.409,A -85,B 0,C 180,E1 -8012.629,E2 -8012.629} C_VEL
LIN {X 0,Y 459.6,Z 475.487,A -85,B 0,C 180,E1 -8013.946,E2 -8013.946} C_VEL
LIN {X 0,Y 459.651,Z 472.828,A -85,B 0,C 180,E1 -8014.824,E2 -8014.824} C_VEL
LIN {X 0,Y 459.769,Z 467.621,A -85,B 0,C 180,E1 -8016.142,E2 -8016.142} C_VEL
LIN {X 0,Y 459.977,Z 460.765,A -85,B 0,C 180,E1 -8017.462,E2 -8017.462} C_VEL
LIN {X 0,Y 460.259,Z 453.273,A -85,B 0,C 180,E1 -8018.562,E2 -8018.562} C_VEL
LIN {X 0,Y 460.584,Z 445.888,A -85,B 0,C 180,E1 -8019.441,E2 -8019.441} C_VEL
LIN {X 0,Y 460.923,Z 437.981,A -85,B 0,C 180,E1 -8020.21,E2 -8020.21} C_VEL
LIN {X 0,Y 461.242,Z 429.629,A -85,B 0,C 180,E1 -8020.868,E2 -8020.868} C_VEL
LIN {X 0,Y 461.617,Z 418.965,A -85,B 0,C 180,E1 -8021.526,E2 -8021.526} C_VEL
LIN {X 0,Y 461.901,Z 407.361,A -85,B 0,C 180,E1 -8022.02,E2 -8022.02} C_VEL
LIN {X 0,Y 462.225,Z 397.665,A -85,B 0,C 180,E1 -8022.29,E2 -8022.29} C_VEL
LIN {X 0,Y 462.533,Z 336.585,A -85,B 0,C 180,E1 -8023.275,E2 -8023.275} C_VEL
LIN {X 0,Y 460.399,Z 320.128,A -85,B 0,C 180,E1 -8023.624,E2 -8023.624} C_VEL
LIN {X 0,Y 460.864,Z 305.592,A -85,B 0,C 180,E1 -8026.591,E2 -8026.591} C_VEL
LIN {X 0,Y 461.417,Z 289.981,A -85,B 0,C 180,E1 -8029.809,E2 -8029.809} C_VEL
LIN {X 0,Y 461.658,Z 279.406,A -85,B 0,C 180,E1 -8032.019,E2 -8032.019} C_VEL
LIN {X 0,Y 460.558,Z 272.93,A -85,B 0,C 180,E1 -8033.491,E2 -8033.491} C_VEL
LIN {X 0,Y 460.516,Z 272.935,A -85,B 0,C 180,E1 -8036.267,E2 -8036.267} C_VEL
LIN {X 0,Y 460.516,Z 272.934,A -85,B 0,C 180,E1 -8039.232,E2 -8039.232} C_VEL
LIN {X 0,Y 460.525,Z 272.93,A -85,B 0,C 180,E1 -8042.284,E2 -8042.284} C_VEL
LIN {X 0,Y 460.503,Z 272.935,A -85,B 0,C 180,E1 -8045.445,E2 -8045.445} C_VEL
LIN {X 0,Y 460.532,Z 272.936,A -85,B 0,C 180,E1 -8048.896,E2 -8048.896} C_VEL
LIN {X 0,Y 460.496,Z 272.932,A -85,B 0,C 180,E1 -8052.183,E2 -8052.183} C_VEL
LIN {X 0,Y 460.506,Z 272.937,A -85,B 0,C 180,E1 -8055.41,E2 -8055.41} C_VEL
LIN {X 0,Y 460.523,Z 272.927,A -85,B 0,C 180,E1 -8058.397,E2 -8058.397} C_VEL
LIN {X 0,Y 460.509,Z 272.935,A -85,B 0,C 180,E1 -8061.265,E2 -8061.265} C_VEL
LIN {X 0,Y 460.502,Z 272.931,A -85,B 0,C 180,E1 -8064.554,E2 -8064.554} C_VEL
LIN {X 0,Y 460.52,Z 272.931,A -85,B 0,C 180,E1 -8067.715,E2 -8067.715} C_VEL
LIN {X 0,Y 460.527,Z 272.927,A -85,B 0,C 180,E1 -8070.768,E2 -8070.768} C_VEL
LIN {X 0,Y 460.544,Z 272.925,A -85,B 0,C 180,E1 -8073.734,E2 -8073.734} C_VEL
LIN {X 0,Y 460.532,Z 272.926,A -85,B 0,C 180,E1 -8076.623,E2 -8076.623} C_VEL
LIN {X 0,Y 460.538,Z 272.923,A -85,B 0,C 180,E1 -8079.452,E2 -8079.452} C_VEL
LIN {X 0,Y 460.544,Z 272.933,A -85,B 0,C 180,E1 -8082.23,E2 -8082.23} C_VEL
LIN {X 0,Y 460.55,Z 272.922,A -85,B 0,C 180,E1 -8084.964,E2 -8084.964} C_VEL
LIN {X 0,Y 460.6,Z 272.924,A -85,B 0,C 180,E1 -8088.559,E2 -8088.559} C_VEL
LIN {X 0,Y 460.682,Z 272.906,A -85,B 0,C 180,E1 -8092.108,E2 -8092.108} C_VEL
LIN {X 0,Y 460.683,Z 272.913,A -85,B 0,C 180,E1 -8094.748,E2 -8094.748} C_VEL
LIN {X 0,Y 460.786,Z 272.894,A -85,B 0,C 180,E1 -8097.378,E2 -8097.378} C_VEL
LIN {X 0,Y 460.837,Z 272.888,A -85,B 0,C 180,E1 -8100,E2 -8100} C_VEL
LIN {X 0,Y 460.786,Z 272.893,A -85,B 0,C 180,E1 -8102.623,E2 -8102.623} C_VEL
LIN {X 0,Y 460.673,Z 272.908,A -85,B 0,C 180,E1 -8106.131,E2 -8106.131} C_VEL
LIN {X 0,Y 460.615,Z 272.915,A -85,B 0,C 180,E1 -8108.776,E2 -8108.776} C_VEL
LIN {X 0,Y 460.596,Z 272.915,A -85,B 0,C 180,E1 -8112.335,E2 -8112.335} C_VEL
LIN {X 0,Y 460.588,Z 272.92,A -85,B 0,C 180,E1 -8115.998,E2 -8115.998} C_VEL
LIN {X 0,Y 460.558,Z 272.926,A -85,B 0,C 180,E1 -8118.902,E2 -8118.902} C_VEL
LIN {X 0,Y 460.504,Z 272.935,A -85,B 0,C 180,E1 -8121.486,E2 -8121.486} C_VEL
LIN {X 0,Y 460.532,Z 272.931,A -85,B 0,C 180,E1 -8124.333,E2 -8124.333} C_VEL
LIN {X 0,Y 460.574,Z 272.922,A -85,B 0,C 180,E1 -8127.244,E2 -8127.244} C_VEL
LIN {X 0,Y 460.516,Z 272.934,A -85,B 0,C 180,E1 -8130.24,E2 -8130.24} C_VEL
LIN {X 0,Y 460.52,Z 272.93,A -85,B 0,C 180,E1 -8133.326,E2 -8133.326} C_VEL
LIN {X 0,Y 460.471,Z 272.941,A -85,B 0,C 180,E1 -8136.53,E2 -8136.53} C_VEL
LIN {X 0,Y 460.567,Z 272.927,A -85,B 0,C 180,E1 -8139.859,E2 -8139.859} C_VEL
LIN {X 0,Y 460.616,Z 272.933,A -85,B 0,C 180,E1 -8143.289,E2 -8143.289} C_VEL
LIN {X 0,Y 460.841,Z 277.032,A -85,B 0,C 180,E1 -8144.214,E2 -8144.214} C_VEL
LIN {X 0,Y 460.595,Z 291.658,A -85,B 0,C 180,E1 -8147.457,E2 -8147.457} C_VEL
LIN {X 0,Y 460.518,Z 296.102,A -85,B 0,C 180,E1 -8148.441,E2 -8148.441} C_VEL
LIN {X 0,Y 462.757,Z 309.678,A -85,B 0,C 180,E1 -8148.742,E2 -8148.742} C_VEL
LIN {X 0,Y 462.218,Z 373.22,A -85,B 0,C 180,E1 -8149.763,E2 -8149.763} C_VEL
LIN {X 0,Y 462.035,Z 384.102,A -85,B 0,C 180,E1 -8150.082,E2 -8150.082} C_VEL
LIN {X 0,Y 461.84,Z 394.801,A -85,B 0,C 180,E1 -8150.565,E2 -8150.565} C_VEL
LIN {X 0,Y 461.476,Z 404.167,A -85,B 0,C 180,E1 -8151.143,E2 -8151.143} C_VEL
LIN {X 0,Y 461.12,Z 413.495,A -85,B 0,C 180,E1 -8151.885,E2 -8151.885} C_VEL
LIN {X 0,Y 460.843,Z 420.193,A -85,B 0,C 180,E1 -8152.538,E2 -8152.538} C_VEL
LIN {X 0,Y 460.539,Z 427.058,A -85,B 0,C 180,E1 -8153.342,E2 -8153.342} C_VEL
LIN {X 0,Y 460.358,Z 431.91,A -85,B 0,C 180,E1 -8154.01,E2 -8154.01} C_VEL
LIN {X 0,Y 460.084,Z 438.176,A -85,B 0,C 180,E1 -8155.053,E2 -8155.053} C_VEL
LIN {X 0,Y 459.951,Z 443.274,A -85,B 0,C 180,E1 -8156.108,E2 -8156.108} C_VEL
LIN {X 0,Y 459.787,Z 446.62,A -85,B 0,C 180,E1 -8156.954,E2 -8156.954} C_VEL
LIN {X 0,Y 459.745,Z 448.987,A -85,B 0,C 180,E1 -8157.655,E2 -8157.655} C_VEL
LIN {X 0,Y 459.64,Z 452.093,A -85,B 0,C 180,E1 -8158.899,E2 -8158.899} C_VEL
LIN {X 0,Y 459.523,Z 453.544,A -85,B 0,C 180,E1 -8159.689,E2 -8159.689} C_VEL
LIN {X 0,Y 459.442,Z 454.719,A -85,B 0,C 180,E1 -8160.693,E2 -8160.693} C_VEL
LIN {X 0,Y 459.415,Z 455.235,A -85,B 0,C 180,E1 -8161.692,E2 -8161.692} C_VEL
LIN {X 0,Y 459.427,Z 455.117,A -85,B 0,C 180,E1 -8162.684,E2 -8162.684} C_VEL
LIN {X 0,Y 459.453,Z 453.679,A -85,B 0,C 180,E1 -8164.213,E2 -8164.213} C_VEL
LIN {X 0,Y 458.849,Z 452.589,A -85,B 0,C 180,E1 -8164.935,E2 -8164.935} C_VEL
LIN {X 0,Y 456.12,Z 450.122,A -85,B 0,C 180,E1 -8166.09,E2 -8166.09} C_VEL
LIN {X 0,Y 453.822,Z 447.462,A -85,B 0,C 180,E1 -8166.993,E2 -8166.993} C_VEL
LIN {X 0,Y 452.872,Z 445.018,A -85,B 0,C 180,E1 -8167.667,E2 -8167.667} C_VEL
LIN {X 0,Y 452.816,Z 444.074,A -85,B 0,C 180,E1 -8167.889,E2 -8167.889} C_VEL
LIN {X 0,Y 452.962,Z 439.722,A -85,B 0,C 180,E1 -8168.843,E2 -8168.843} C_VEL
LIN {X 0,Y 453.215,Z 434.273,A -85,B 0,C 180,E1 -8169.817,E2 -8169.817} C_VEL
LIN {X 0,Y 453.514,Z 427.545,A -85,B 0,C 180,E1 -8170.798,E2 -8170.798} C_VEL
LIN {X 0,Y 453.803,Z 420.806,A -85,B 0,C 180,E1 -8171.607,E2 -8171.607} C_VEL
LIN {X 0,Y 454.118,Z 413.654,A -85,B 0,C 180,E1 -8172.319,E2 -8172.319} C_VEL
LIN {X 0,Y 454.476,Z 405.433,A -85,B 0,C 180,E1 -8172.989,E2 -8172.989} C_VEL
LIN {X 0,Y 454.764,Z 395.9,A -85,B 0,C 180,E1 -8173.605,E2 -8173.605} C_VEL
LIN {X 0,Y 455.046,Z 383.555,A -85,B 0,C 180,E1 -8174.176,E2 -8174.176} C_VEL
LIN {X 0,Y 455.301,Z 373.496,A -85,B 0,C 180,E1 -8174.472,E2 -8174.472} C_VEL
LIN {X 0,Y 455.546,Z 338.738,A -85,B 0,C 180,E1 -8175.053,E2 -8175.053} C_VEL
LIN {X 0,Y 455.672,Z 309.961,A -85,B 0,C 180,E1 -8175.514,E2 -8175.514} C_VEL
LIN {X 0,Y 453.482,Z 296.603,A -85,B 0,C 180,E1 -8175.815,E2 -8175.815} C_VEL
LIN {X 0,Y 453.829,Z 284.331,A -85,B 0,C 180,E1 -8178.839,E2 -8178.839} C_VEL
LIN {X 0,Y 453.956,Z 277.083,A -85,B 0,C 180,E1 -8180.645,E2 -8180.645} C_VEL
LIN {X 0,Y 453.672,Z 273.79,A -85,B 0,C 180,E1 -8181.537,E2 -8181.537} C_VEL
LIN {X 0,Y 453.668,Z 273.781,A -85,B 0,C 180,E1 -8184.667,E2 -8184.667} C_VEL
LIN {X 0,Y 453.745,Z 273.774,A -85,B 0,C 180,E1 -8187.337,E2 -8187.337} C_VEL
LIN {X 0,Y 453.825,Z 273.769,A -85,B 0,C 180,E1 -8190,E2 -8190} C_VEL
LIN {X 0,Y 453.746,Z 273.773,A -85,B 0,C 180,E1 -8192.663,E2 -8192.663} C_VEL
LIN {X 0,Y 453.652,Z 273.791,A -85,B 0,C 180,E1 -8196.225,E2 -8196.225} C_VEL
LIN {X 0,Y 453.592,Z 273.792,A -85,B 0,C 180,E1 -8198.913,E2 -8198.913} C_VEL
LIN {X 0,Y 453.565,Z 273.8,A -85,B 0,C 180,E1 -8202.528,E2 -8202.528} C_VEL
LIN {X 0,Y 453.545,Z 273.801,A -85,B 0,C 180,E1 -8206.195,E2 -8206.195} C_VEL
LIN {X 0,Y 453.517,Z 273.803,A -85,B 0,C 180,E1 -8209.039,E2 -8209.039} C_VEL
LIN {X 0,Y 453.476,Z 273.805,A -85,B 0,C 180,E1 -8211.835,E2 -8211.835} C_VEL
LIN {X 0,Y 453.506,Z 273.81,A -85,B 0,C 180,E1 -8214.734,E2 -8214.734} C_VEL
LIN {X 0,Y 453.531,Z 273.798,A -85,B 0,C 180,E1 -8217.959,E2 -8217.959} C_VEL
LIN {X 0,Y 453.462,Z 273.809,A -85,B 0,C 180,E1 -8221.524,E2 -8221.524} C_VEL
LIN {X 0,Y 453.479,Z 273.808,A -85,B 0,C 180,E1 -8224.775,E2 -8224.775} C_VEL
LIN {X 0,Y 453.46,Z 273.807,A -85,B 0,C 180,E1 -8228.311,E2 -8228.311} C_VEL
LIN {X 0,Y 453.489,Z 273.804,A -85,B 0,C 180,E1 -8230.608,E2 -8230.608} C_VEL
LIN {X 0,Y 453.451,Z 273.814,A -85,B 0,C 180,E1 -8233.243,E2 -8233.243} C_VEL
LIN {X 0,Y 453.471,Z 273.811,A -85,B 0,C 180,E1 -8235.779,E2 -8235.779} C_VEL
LIN {X 0,Y 453.49,Z 273.805,A -85,B 0,C 180,E1 -8238.21,E2 -8238.21} C_VEL
LIN {X 0,Y 453.519,Z 273.8,A -85,B 0,C 180,E1 -8240.787,E2 -8240.787} C_VEL
LIN {X 0,Y 453.449,Z 273.816,A -85,B 0,C 180,E1 -8243.917,E2 -8243.917} C_VEL
LIN {X 0,Y 453.474,Z 273.806,A -85,B 0,C 180,E1 -8247.15,E2 -8247.15} C_VEL
LIN {X 0,Y 453.505,Z 273.807,A -85,B 0,C 180,E1 -8250.27,E2 -8250.27} C_VEL
LIN {X 0,Y 453.504,Z 273.802,A -85,B 0,C 180,E1 -8253.294,E2 -8253.294} C_VEL
LIN {X 0,Y 453.493,Z 273.812,A -85,B 0,C 180,E1 -8256.238,E2 -8256.238} C_VEL
LIN {X 0,Y 453.471,Z 273.806,A -85,B 0,C 180,E1 -8259.117,E2 -8259.117} C_VEL
LIN {X 0,Y 453.499,Z 273.804,A -85,B 0,C 180,E1 -8261.944,E2 -8261.944} C_VEL
LIN {X 0,Y 453.527,Z 273.805,A -85,B 0,C 180,E1 -8264.726,E2 -8264.726} C_VEL
LIN {X 0,Y 453.547,Z 273.801,A -85,B 0,C 180,E1 -8268.379,E2 -8268.379} C_VEL
LIN {X 0,Y 453.639,Z 273.785,A -85,B 0,C 180,E1 -8271.985,E2 -8271.985} C_VEL
LIN {X 0,Y 453.654,Z 273.788,A -85,B 0,C 180,E1 -8274.666,E2 -8274.666} C_VEL
LIN {X 0,Y 453.751,Z 273.775,A -85,B 0,C 180,E1 -8277.337,E2 -8277.337} C_VEL
LIN {X 0,Y 453.808,Z 273.764,A -85,B 0,C 180,E1 -8280,E2 -8280} C_VEL
LIN {X 0,Y 453.731,Z 273.775,A -85,B 0,C 180,E1 -8282.663,E2 -8282.663} C_VEL
LIN {X 0,Y 453.658,Z 273.783,A -85,B 0,C 180,E1 -8286.225,E2 -8286.225} C_VEL
LIN {X 0,Y 453.58,Z 273.794,A -85,B 0,C 180,E1 -8288.913,E2 -8288.913} C_VEL
LIN {X 0,Y 453.59,Z 273.791,A -85,B 0,C 180,E1 -8292.551,E2 -8292.551} C_VEL
LIN {X 0,Y 453.533,Z 273.8,A -85,B 0,C 180,E1 -8296.196,E2 -8296.196} C_VEL
LIN {X 0,Y 453.507,Z 273.802,A -85,B 0,C 180,E1 -8299.041,E2 -8299.041} C_VEL
LIN {X 0,Y 453.465,Z 273.815,A -85,B 0,C 180,E1 -8301.837,E2 -8301.837} C_VEL
LIN {X 0,Y 453.503,Z 273.802,A -85,B 0,C 180,E1 -8304.735,E2 -8304.735} C_VEL
LIN {X 0,Y 453.52,Z 273.806,A -85,B 0,C 180,E1 -8307.96,E2 -8307.96} C_VEL
LIN {X 0,Y 453.455,Z 273.809,A -85,B 0,C 180,E1 -8311.526,E2 -8311.526} C_VEL
LIN {X 0,Y 453.479,Z 273.808,A -85,B 0,C 180,E1 -8314.778,E2 -8314.778} C_VEL
LIN {X 0,Y 453.451,Z 273.815,A -85,B 0,C 180,E1 -8318.313,E2 -8318.313} C_VEL
LIN {X 0,Y 453.485,Z 273.812,A -85,B 0,C 180,E1 -8320.61,E2 -8320.61} C_VEL
LIN {X 0,Y 453.446,Z 273.81,A -85,B 0,C 180,E1 -8323.245,E2 -8323.245} C_VEL
LIN {X 0,Y 453.452,Z 273.808,A -85,B 0,C 180,E1 -8325.779,E2 -8325.779} C_VEL
LIN {X 0,Y 453.487,Z 273.806,A -85,B 0,C 180,E1 -8329.41,E2 -8329.41} C_VEL
LIN {X 0,Y 453.443,Z 273.81,A -85,B 0,C 180,E1 -8332.228,E2 -8332.228} C_VEL
LIN {X 0,Y 453.477,Z 273.811,A -85,B 0,C 180,E1 -8335.225,E2 -8335.225} C_VEL
LIN {X 0,Y 453.46,Z 273.808,A -85,B 0,C 180,E1 -8338.476,E2 -8338.476} C_VEL
LIN {X 0,Y 453.488,Z 273.813,A -85,B 0,C 180,E1 -8341.288,E2 -8341.288} C_VEL
LIN {X 0,Y 453.491,Z 273.806,A -85,B 0,C 180,E1 -8344.284,E2 -8344.284} C_VEL
LIN {X 0,Y 453.517,Z 273.866,A -85,B 0,C 180,E1 -8346.179,E2 -8346.179} C_VEL
LIN {X 0,Y 454.846,Z 281.755,A -85,B 0,C 180,E1 -8347.984,E2 -8347.984} C_VEL
LIN {X 0,Y 454.376,Z 293.191,A -85,B 0,C 180,E1 -8350.456,E2 -8350.456} C_VEL
LIN {X 0,Y 453.811,Z 308.94,A -85,B 0,C 180,E1 -8353.814,E2 -8353.814} C_VEL
LIN {X 0,Y 453.424,Z 320.589,A -85,B 0,C 180,E1 -8356.235,E2 -8356.235} C_VEL
LIN {X 0,Y 455.635,Z 338.932,A -85,B 0,C 180,E1 -8356.597,E2 -8356.597} C_VEL
LIN {X 0,Y 455.219,Z 397.214,A -85,B 0,C 180,E1 -8357.546,E2 -8357.546} C_VEL
LIN {X 0,Y 454.944,Z 407.052,A -85,B 0,C 180,E1 -8357.822,E2 -8357.822} C_VEL
LIN {X 0,Y 454.666,Z 417.003,A -85,B 0,C 180,E1 -8358.238,E2 -8358.238} C_VEL
LIN {X 0,Y 454.28,Z 427.571,A -85,B 0,C 180,E1 -8358.85,E2 -8358.85} C_VEL
LIN {X 0,Y 453.919,Z 437.521,A -85,B 0,C 180,E1 -8359.631,E2 -8359.631} C_VEL
LIN {X 0,Y 453.57,Z 445.486,A -85,B 0,C 180,E1 -8360.412,E2 -8360.412} C_VEL
LIN {X 0,Y 453.234,Z 452.923,A -85,B 0,C 180,E1 -8361.305,E2 -8361.305} C_VEL
LIN {X 0,Y 452.905,Z 460.464,A -85,B 0,C 180,E1 -8362.421,E2 -8362.421} C_VEL
LIN {X 0,Y 452.709,Z 467.37,A -85,B 0,C 180,E1 -8363.762,E2 -8363.762} C_VEL
LIN {X 0,Y 452.583,Z 472.589,A -85,B 0,C 180,E1 -8365.101,E2 -8365.101} C_VEL
LIN {X 0,Y 452.5,Z 475.264,A -85,B 0,C 180,E1 -8365.992,E2 -8365.992} C_VEL
LIN {X 0,Y 452.514,Z 478.195,A -85,B 0,C 180,E1 -8367.33,E2 -8367.33} C_VEL
LIN {X 0,Y 452.435,Z 479.463,A -85,B 0,C 180,E1 -8368.22,E2 -8368.22} C_VEL
LIN {X 0,Y 452.426,Z 480.256,A -85,B 0,C 180,E1 -8369.11,E2 -8369.11} C_VEL
LIN {X 0,Y 452.433,Z 480.553,A -85,B 0,C 180,E1 -8370,E2 -8370} C_VEL
LIN {X 0,Y 452.426,Z 480.255,A -85,B 0,C 180,E1 -8370.89,E2 -8370.89} C_VEL
LIN {X 0,Y 452.435,Z 479.475,A -85,B 0,C 180,E1 -8371.78,E2 -8371.78} C_VEL
LIN {X 0,Y 452.514,Z 478.22,A -85,B 0,C 180,E1 -8372.67,E2 -8372.67} C_VEL
LIN {X 0,Y 452.5,Z 475.299,A -85,B 0,C 180,E1 -8374.008,E2 -8374.008} C_VEL
LIN {X 0,Y 452.583,Z 472.643,A -85,B 0,C 180,E1 -8374.899,E2 -8374.899} C_VEL
LIN {X 0,Y 452.681,Z 467.437,A -85,B 0,C 180,E1 -8376.239,E2 -8376.239} C_VEL
LIN {X 0,Y 452.884,Z 461.842,A -85,B 0,C 180,E1 -8377.355,E2 -8377.355} C_VEL
LIN {X 0,Y 453.151,Z 454.802,A -85,B 0,C 180,E1 -8378.472,E2 -8378.472} C_VEL
LIN {X 0,Y 453.542,Z 446.742,A -85,B 0,C 180,E1 -8379.476,E2 -8379.476} C_VEL
LIN {X 0,Y 453.869,Z 439.049,A -85,B 0,C 180,E1 -8380.257,E2 -8380.257} C_VEL
LIN {X 0,Y 454.211,Z 430.973,A -85,B 0,C 180,E1 -8380.926,E2 -8380.926} C_VEL
LIN {X 0,Y 454.504,Z 422.61,A -85,B 0,C 180,E1 -8381.483,E2 -8381.483} C_VEL
LIN {X 0,Y 454.773,Z 414.083,A -85,B 0,C 180,E1 -8381.928,E2 -8381.928} C_VEL
LIN {X 0,Y 455.092,Z 403.936,A -85,B 0,C 180,E1 -8382.316,E2 -8382.316} C_VEL
LIN {X 0,Y 455.391,Z 391.503,A -85,B 0,C 180,E1 -8382.603,E2 -8382.603} C_VEL
LIN {X 0,Y 455.553,Z 336.691,A -85,B 0,C 180,E1 -8383.482,E2 -8383.482} C_VEL
LIN {X 0,Y 453.388,Z 319.952,A -85,B 0,C 180,E1 -8383.839,E2 -8383.839} C_VEL
LIN {X 0,Y 453.897,Z 304.182,A -85,B 0,C 180,E1 -8387.108,E2 -8387.108} C_VEL
LIN {X 0,Y 454.512,Z 288.675,A -85,B 0,C 180,E1 -8390.359,E2 -8390.359} C_VEL
LIN {X 0,Y 454.697,Z 281.092,A -85,B 0,C 180,E1 -8391.969,E2 -8391.969} C_VEL
LIN {X 0,Y 453.497,Z 273.81,A -85,B 0,C 180,E1 -8393.64,E2 -8393.64} C_VEL
LIN {X 0,Y 453.452,Z 273.816,A -85,B 0,C 180,E1 -8396.709,E2 -8396.709} C_VEL
LIN {X 0,Y 453.464,Z 273.811,A -85,B 0,C 180,E1 -8399.783,E2 -8399.783} C_VEL
LIN {X 0,Y 453.479,Z 273.811,A -85,B 0,C 180,E1 -8403.187,E2 -8403.187} C_VEL
LIN {X 0,Y 453.447,Z 273.812,A -85,B 0,C 180,E1 -8406.298,E2 -8406.298} C_VEL
LIN {X 0,Y 453.476,Z 273.814,A -85,B 0,C 180,E1 -8409.45,E2 -8409.45} C_VEL
LIN {X 0,Y 453.452,Z 273.811,A -85,B 0,C 180,E1 -8411.931,E2 -8411.931} C_VEL
LIN {X 0,Y 453.476,Z 273.813,A -85,B 0,C 180,E1 -8415.47,E2 -8415.47} C_VEL
LIN {X 0,Y 453.471,Z 273.806,A -85,B 0,C 180,E1 -8418.208,E2 -8418.208} C_VEL
LIN {X 0,Y 453.462,Z 273.809,A -85,B 0,C 180,E1 -8420.796,E2 -8420.796} C_VEL
LIN {X 0,Y 453.446,Z 273.815,A -85,B 0,C 180,E1 -8423.917,E2 -8423.917} C_VEL
LIN {X 0,Y 453.472,Z 273.805,A -85,B 0,C 180,E1 -8427.15,E2 -8427.15} C_VEL
LIN {X 0,Y 453.463,Z 273.81,A -85,B 0,C 180,E1 -8430.268,E2 -8430.268} C_VEL
LIN {X 0,Y 453.489,Z 273.799,A -85,B 0,C 180,E1 -8433.293,E2 -8433.293} C_VEL
LIN {X 0,Y 453.485,Z 273.808,A -85,B 0,C 180,E1 -8436.238,E2 -8436.238} C_VEL
LIN {X 0,Y 453.469,Z 273.803,A -85,B 0,C 180,E1 -8439.117,E2 -8439.117} C_VEL
LIN {X 0,Y 453.497,Z 273.807,A -85,B 0,C 180,E1 -8441.944,E2 -8441.944} C_VEL
LIN {X 0,Y 453.525,Z 273.8,A -85,B 0,C 180,E1 -8444.726,E2 -8444.726} C_VEL
LIN {X 0,Y 453.548,Z 273.804,A -85,B 0,C 180,E1 -8448.379,E2 -8448.379} C_VEL
LIN {X 0,Y 453.639,Z 273.782,A -85,B 0,C 180,E1 -8451.985,E2 -8451.985} C_VEL
LIN {X 0,Y 453.656,Z 273.789,A -85,B 0,C 180,E1 -8454.667,E2 -8454.667} C_VEL
LIN {X 0,Y 453.73,Z 273.773,A -85,B 0,C 180,E1 -8457.337,E2 -8457.337} C_VEL
LIN {X 0,Y 453.808,Z 273.763,A -85,B 0,C 180,E1 -8460,E2 -8460} C_VEL
LIN {X 0,Y 453.731,Z 273.772,A -85,B 0,C 180,E1 -8462.663,E2 -8462.663} C_VEL
LIN {X 0,Y 453.639,Z 273.784,A -85,B 0,C 180,E1 -8466.226,E2 -8466.226} C_VEL
LIN {X 0,Y 453.579,Z 273.793,A -85,B 0,C 180,E1 -8468.914,E2 -8468.914} C_VEL
LIN {X 0,Y 453.551,Z 273.792,A -85,B 0,C 180,E1 -8472.529,E2 -8472.529} C_VEL
LIN {X 0,Y 453.533,Z 273.797,A -85,B 0,C 180,E1 -8476.196,E2 -8476.196} C_VEL
LIN {X 0,Y 453.508,Z 273.805,A -85,B 0,C 180,E1 -8479.041,E2 -8479.041} C_VEL
LIN {X 0,Y 453.465,Z 273.817,A -85,B 0,C 180,E1 -8481.837,E2 -8481.837} C_VEL
LIN {X 0,Y 453.504,Z 273.804,A -85,B 0,C 180,E1 -8484.735,E2 -8484.735} C_VEL
LIN {X 0,Y 453.528,Z 273.807,A -85,B 0,C 180,E1 -8487.962,E2 -8487.962} C_VEL
LIN {X 0,Y 453.473,Z 273.807,A -85,B 0,C 180,E1 -8490.76,E2 -8490.76} C_VEL
LIN {X 0,Y 453.469,Z 273.813,A -85,B 0,C 180,E1 -8493.913,E2 -8493.913} C_VEL
LIN {X 0,Y 453.463,Z 273.81,A -85,B 0,C 180,E1 -8497.189,E2 -8497.189} C_VEL
LIN {X 0,Y 453.521,Z 273.803,A -85,B 0,C 180,E1 -8499.447,E2 -8499.447} C_VEL
LIN {X 0,Y 453.602,Z 273.911,A -85,B 0,C 180,E1 -8503.185,E2 -8503.185} C_VEL
LIN {X 0,Y 453.855,Z 278.241,A -85,B 0,C 180,E1 -8504.173,E2 -8504.173} C_VEL
LIN {X 0,Y 453.577,Z 292.163,A -85,B 0,C 180,E1 -8507.302,E2 -8507.302} C_VEL
LIN {X 0,Y 453.527,Z 296.26,A -85,B 0,C 180,E1 -8508.216,E2 -8508.216} C_VEL
LIN {X 0,Y 455.869,Z 310.136,A -85,B 0,C 180,E1 -8508.535,E2 -8508.535} C_VEL
LIN {X 0,Y 455.314,Z 373.151,A -85,B 0,C 180,E1 -8509.564,E2 -8509.564} C_VEL
LIN {X 0,Y 455.151,Z 383.324,A -85,B 0,C 180,E1 -8509.861,E2 -8509.861} C_VEL
LIN {X 0,Y 454.875,Z 395.427,A -85,B 0,C 180,E1 -8510.409,E2 -8510.409} C_VEL
LIN {X 0,Y 454.544,Z 404.036,A -85,B 0,C 180,E1 -8510.947,E2 -8510.947} C_VEL
LIN {X 0,Y 454.21,Z 412.579,A -85,B 0,C 180,E1 -8511.623,E2 -8511.623} C_VEL
LIN {X 0,Y 453.867,Z 420.124,A -85,B 0,C 180,E1 -8512.357,E2 -8512.357} C_VEL
LIN {X 0,Y 453.591,Z 426.228,A -85,B 0,C 180,E1 -8513.068,E2 -8513.068} C_VEL
LIN {X 0,Y 453.329,Z 432.271,A -85,B 0,C 180,E1 -8513.907,E2 -8513.907} C_VEL
LIN {X 0,Y 453.033,Z 438.542,A -85,B 0,C 180,E1 -8514.972,E2 -8514.972} C_VEL
LIN {X 0,Y 452.892,Z 443.59,A -85,B 0,C 180,E1 -8516.039,E2 -8516.039} C_VEL
LIN {X 0,Y 452.678,Z 447.55,A -85,B 0,C 180,E1 -8517.087,E2 -8517.087} C_VEL
LIN {X 0,Y 452.629,Z 450.624,A -85,B 0,C 180,E1 -8518.136,E2 -8518.136} C_VEL
LIN {X 0,Y 452.521,Z 452.877,A -85,B 0,C 180,E1 -8519.17,E2 -8519.17} C_VEL
LIN {X 0,Y 452.377,Z 454.691,A -85,B 0,C 180,E1 -8520.459,E2 -8520.459} C_VEL
LIN {X 0,Y 452.317,Z 455.265,A -85,B 0,C 180,E1 -8521.206,E2 -8521.206} C_VEL
LIN {X 0,Y 452.321,Z 455.445,A -85,B 0,C 180,E1 -8522.331,E2 -8522.331} C_VEL
LIN {X 0,Y 452.325,Z 455.075,A -85,B 0,C 180,E1 -8523.22,E2 -8523.22} C_VEL
LIN {X 0,Y 452.387,Z 453.893,A -85,B 0,C 180,E1 -8524.297,E2 -8524.297} C_VEL
LIN {X 0,Y 452.577,Z 451.15,A -85,B 0,C 180,E1 -8525.701,E2 -8525.701} C_VEL
LIN {X 0,Y 452.676,Z 448.194,A -85,B 0,C 180,E1 -8526.763,E2 -8526.763} C_VEL
LIN {X 0,Y 452.816,Z 444.074,A -85,B 0,C 180,E1 -8527.889,E2 -8527.889} C_VEL
LIN {X 0,Y 452.235,Z 441.337,A -85,B 0,C 180,E1 -8528.538,E2 -8528.538} C_VEL
LIN {X 0,Y 449.572,Z 436.28,A -85,B 0,C 180,E1 -8529.567,E2 -8529.567} C_VEL
LIN {X 0,Y 446.992,Z 430.508,A -85,B 0,C 180,E1 -8530.544,E2 -8530.544} C_VEL
LIN {X 0,Y 446.559,Z 426.403,A -85,B 0,C 180,E1 -8531.107,E2 -8531.107} C_VEL
LIN {X 0,Y 446.976,Z 417.387,A -85,B 0,C 180,E1 -8532.146,E2 -8532.146} C_VEL
LIN {X 0,Y 447.357,Z 408.621,A -85,B 0,C 180,E1 -8532.929,E2 -8532.929} C_VEL
LIN {X 0,Y 447.68,Z 399.293,A -85,B 0,C 180,E1 -8533.586,E2 -8533.586} C_VEL
LIN {X 0,Y 447.956,Z 390.548,A -85,B 0,C 180,E1 -8534.065,E2 -8534.065} C_VEL
LIN {X 0,Y 448.158,Z 381.03,A -85,B 0,C 180,E1 -8534.451,E2 -8534.451} C_VEL
LIN {X 0,Y 448.355,Z 370.97,A -85,B 0,C 180,E1 -8534.72,E2 -8534.72} C_VEL
LIN {X 0,Y 448.707,Z 310.247,A -85,B 0,C 180,E1 -8535.719,E2 -8535.719} C_VEL
LIN {X 0,Y 446.476,Z 296.805,A -85,B 0,C 180,E1 -8536.024,E2 -8536.024} C_VEL
LIN {X 0,Y 446.859,Z 284.397,A -85,B 0,C 180,E1 -8539.122,E2 -8539.122} C_VEL
LIN {X 0,Y 446.892,Z 277.164,A -85,B 0,C 180,E1 -8540.952,E2 -8540.952} C_VEL
LIN {X 0,Y 446.636,Z 274.666,A -85,B 0,C 180,E1 -8541.631,E2 -8541.631} C_VEL
LIN {X 0,Y 446.643,Z 274.657,A -85,B 0,C 180,E1 -8544.583,E2 -8544.583} C_VEL
LIN {X 0,Y 446.666,Z 274.657,A -85,B 0,C 180,E1 -8548.197,E2 -8548.197} C_VEL
LIN {X 0,Y 446.795,Z 274.645,A -85,B 0,C 180,E1 -8550,E2 -8550} C_VEL
LIN {X 0,Y 446.693,Z 274.651,A -85,B 0,C 180,E1 -8552.705,E2 -8552.705} C_VEL
LIN {X 0,Y 446.621,Z 274.665,A -85,B 0,C 180,E1 -8556.324,E2 -8556.324} C_VEL
LIN {X 0,Y 446.538,Z 274.67,A -85,B 0,C 180,E1 -8559.055,E2 -8559.055} C_VEL
LIN {X 0,Y 446.523,Z 274.675,A -85,B 0,C 180,E1 -8562.729,E2 -8562.729} C_VEL
LIN {X 0,Y 446.496,Z 274.68,A -85,B 0,C 180,E1 -8566.227,E2 -8566.227} C_VEL
LIN {X 0,Y 446.469,Z 274.679,A -85,B 0,C 180,E1 -8569.303,E2 -8569.303} C_VEL
LIN {X 0,Y 446.418,Z 274.687,A -85,B 0,C 180,E1 -8572.199,E2 -8572.199} C_VEL
LIN {X 0,Y 446.448,Z 274.684,A -85,B 0,C 180,E1 -8575.152,E2 -8575.152} C_VEL
LIN {X 0,Y 446.483,Z 274.677,A -85,B 0,C 180,E1 -8578.178,E2 -8578.178} C_VEL
LIN {X 0,Y 446.415,Z 274.685,A -85,B 0,C 180,E1 -8581.774,E2 -8581.774} C_VEL
LIN {X 0,Y 446.419,Z 274.686,A -85,B 0,C 180,E1 -8584.523,E2 -8584.523} C_VEL
LIN {X 0,Y 446.411,Z 274.686,A -85,B 0,C 180,E1 -8588.078,E2 -8588.078} C_VEL
LIN {X 0,Y 446.422,Z 274.687,A -85,B 0,C 180,E1 -8590.917,E2 -8590.917} C_VEL
LIN {X 0,Y 446.396,Z 274.691,A -85,B 0,C 180,E1 -8593.845,E2 -8593.845} C_VEL
LIN {X 0,Y 446.441,Z 274.682,A -85,B 0,C 180,E1 -8596.396,E2 -8596.396} C_VEL
LIN {X 0,Y 446.461,Z 274.686,A -85,B 0,C 180,E1 -8599.804,E2 -8599.804} C_VEL
LIN {X 0,Y 446.424,Z 274.687,A -85,B 0,C 180,E1 -8602.123,E2 -8602.123} C_VEL
LIN {X 0,Y 446.422,Z 274.687,A -85,B 0,C 180,E1 -8605.476,E2 -8605.476} C_VEL
LIN {X 0,Y 446.41,Z 274.686,A -85,B 0,C 180,E1 -8608.699,E2 -8608.699} C_VEL
LIN {X 0,Y 446.475,Z 274.682,A -85,B 0,C 180,E1 -8611.821,E2 -8611.821} C_VEL
LIN {X 0,Y 446.448,Z 274.682,A -85,B 0,C 180,E1 -8614.847,E2 -8614.847} C_VEL
LIN {X 0,Y 446.437,Z 274.69,A -85,B 0,C 180,E1 -8618.244,E2 -8618.244} C_VEL
LIN {X 0,Y 446.445,Z 274.681,A -85,B 0,C 180,E1 -8621.649,E2 -8621.649} C_VEL
LIN {X 0,Y 446.495,Z 274.682,A -85,B 0,C 180,E1 -8624.479,E2 -8624.479} C_VEL
LIN {X 0,Y 446.505,Z 274.676,A -85,B 0,C 180,E1 -8628.193,E2 -8628.193} C_VEL
LIN {X 0,Y 446.588,Z 274.663,A -85,B 0,C 180,E1 -8631.857,E2 -8631.857} C_VEL
LIN {X 0,Y 446.628,Z 274.662,A -85,B 0,C 180,E1 -8634.582,E2 -8634.582} C_VEL
LIN {X 0,Y 446.695,Z 274.654,A -85,B 0,C 180,E1 -8637.295,E2 -8637.295} C_VEL
LIN {X 0,Y 446.779,Z 274.639,A -85,B 0,C 180,E1 -8640,E2 -8640} C_VEL
LIN {X 0,Y 446.679,Z 274.654,A -85,B 0,C 180,E1 -8642.705,E2 -8642.705} C_VEL
LIN {X 0,Y 446.627,Z 274.658,A -85,B 0,C 180,E1 -8646.324,E2 -8646.324} C_VEL
LIN {X 0,Y 446.527,Z 274.674,A -85,B 0,C 180,E1 -8649.055,E2 -8649.055} C_VEL
LIN {X 0,Y 446.521,Z 274.672,A -85,B 0,C 180,E1 -8652.73,E2 -8652.73} C_VEL
LIN {X 0,Y 446.478,Z 274.677,A -85,B 0,C 180,E1 -8656.459,E2 -8656.459} C_VEL
LIN {X 0,Y 446.457,Z 274.682,A -85,B 0,C 180,E1 -8659.304,E2 -8659.304} C_VEL
LIN {X 0,Y 446.406,Z 274.69,A -85,B 0,C 180,E1 -8662.2,E2 -8662.2} C_VEL
LIN {X 0,Y 446.446,Z 274.681,A -85,B 0,C 180,E1 -8665.153,E2 -8665.153} C_VEL
LIN {X 0,Y 446.474,Z 274.685,A -85,B 0,C 180,E1 -8668.179,E2 -8668.179} C_VEL
LIN {X 0,Y 446.408,Z 274.688,A -85,B 0,C 180,E1 -8671.775,E2 -8671.775} C_VEL
LIN {X 0,Y 446.421,Z 274.69,A -85,B 0,C 180,E1 -8674.524,E2 -8674.524} C_VEL
LIN {X 0,Y 446.404,Z 274.69,A -85,B 0,C 180,E1 -8678.08,E2 -8678.08} C_VEL
LIN {X 0,Y 446.42,Z 274.684,A -85,B 0,C 180,E1 -8681.392,E2 -8681.392} C_VEL
LIN {X 0,Y 446.443,Z 274.685,A -85,B 0,C 180,E1 -8685.105,E2 -8685.105} C_VEL
LIN {X 0,Y 446.411,Z 274.691,A -85,B 0,C 180,E1 -8688.609,E2 -8688.609} C_VEL
LIN {X 0,Y 446.433,Z 274.69,A -85,B 0,C 180,E1 -8690.973,E2 -8690.973} C_VEL
LIN {X 0,Y 446.412,Z 274.686,A -85,B 0,C 180,E1 -8694.375,E2 -8694.375} C_VEL
LIN {X 0,Y 446.415,Z 274.687,A -85,B 0,C 180,E1 -8697.639,E2 -8697.639} C_VEL
LIN {X 0,Y 446.432,Z 274.685,A -85,B 0,C 180,E1 -8700.79,E2 -8700.79} C_VEL
LIN {X 0,Y 446.432,Z 274.688,A -85,B 0,C 180,E1 -8703.846,E2 -8703.846} C_VEL
LIN {X 0,Y 446.485,Z 274.715,A -85,B 0,C 180,E1 -8706.021,E2 -8706.021} C_VEL
LIN {X 0,Y 447.828,Z 282.68,A -85,B 0,C 180,E1 -8707.875,E2 -8707.875} C_VEL
LIN {X 0,Y 447.546,Z 291.372,A -85,B 0,C 180,E1 -8709.79,E2 -8709.79} C_VEL
LIN {X 0,Y 446.855,Z 307.638,A -85,B 0,C 180,E1 -8713.32,E2 -8713.32} C_VEL
LIN {X 0,Y 446.371,Z 320.136,A -85,B 0,C 180,E1 -8716,E2 -8716} C_VEL
LIN {X 0,Y 448.728,Z 339.941,A -85,B 0,C 180,E1 -8716.413,E2 -8716.413} C_VEL
LIN {X 0,Y 448.295,Z 396.705,A -85,B 0,C 180,E1 -8717.351,E2 -8717.351} C_VEL
LIN {X 0,Y 448.022,Z 405.824,A -85,B 0,C 180,E1 -8717.602,E2 -8717.602} C_VEL
LIN {X 0,Y 447.71,Z 415.449,A -85,B 0,C 180,E1 -8717.996,E2 -8717.996} C_VEL
LIN {X 0,Y 447.382,Z 425.537,A -85,B 0,C 180,E1 -8718.561,E2 -8718.561} C_VEL
LIN {X 0,Y 446.97,Z 436.018,A -85,B 0,C 180,E1 -8719.354,E2 -8719.354} C_VEL
LIN {X 0,Y 446.619,Z 444.205,A -85,B 0,C 180,E1 -8720.147,E2 -8720.147} C_VEL
LIN {X 0,Y 446.293,Z 450.966,A -85,B 0,C 180,E1 -8720.94,E2 -8720.94} C_VEL
LIN {X 0,Y 445.954,Z 457.375,A -85,B 0,C 180,E1 -8721.846,E2 -8721.846} C_VEL
LIN {X 0,Y 445.787,Z 462.704,A -85,B 0,C 180,E1 -8722.755,E2 -8722.755} C_VEL
LIN {X 0,Y 445.644,Z 467.148,A -85,B 0,C 180,E1 -8723.662,E2 -8723.662} C_VEL
LIN {X 0,Y 445.516,Z 472.373,A -85,B 0,C 180,E1 -8725.023,E2 -8725.023} C_VEL
LIN {X 0,Y 445.407,Z 475.053,A -85,B 0,C 180,E1 -8725.928,E2 -8725.928} C_VEL
LIN {X 0,Y 445.44,Z 477.99,A -85,B 0,C 180,E1 -8727.287,E2 -8727.287} C_VEL
LIN {X 0,Y 445.355,Z 479.262,A -85,B 0,C 180,E1 -8728.191,E2 -8728.191} C_VEL
LIN {X 0,Y 445.336,Z 480.058,A -85,B 0,C 180,E1 -8729.096,E2 -8729.096} C_VEL
LIN {X 0,Y 445.341,Z 480.356,A -85,B 0,C 180,E1 -8730,E2 -8730} C_VEL
LIN {X 0,Y 445.336,Z 480.06,A -85,B 0,C 180,E1 -8730.904,E2 -8730.904} C_VEL
LIN {X 0,Y 445.355,Z 479.283,A -85,B 0,C 180,E1 -8731.809,E2 -8731.809} C_VEL
LIN {X 0,Y 445.44,Z 478.03,A -85,B 0,C 180,E1 -8732.713,E2 -8732.713} C_VEL
LIN {X 0,Y 445.407,Z 475.111,A -85,B 0,C 180,E1 -8734.072,E2 -8734.072} C_VEL
LIN {X 0,Y 445.515,Z 472.457,A -85,B 0,C 180,E1 -8734.977,E2 -8734.977} C_VEL
LIN {X 0,Y 445.616,Z 467.252,A -85,B 0,C 180,E1 -8736.338,E2 -8736.338} C_VEL
LIN {X 0,Y 445.813,Z 461.66,A -85,B 0,C 180,E1 -8737.473,E2 -8737.473} C_VEL
LIN {X 0,Y 446.106,Z 454.628,A -85,B 0,C 180,E1 -8738.607,E2 -8738.607} C_VEL
LIN {X 0,Y 446.508,Z 446.577,A -85,B 0,C 180,E1 -8739.627,E2 -8739.627} C_VEL
LIN {X 0,Y 446.88,Z 438.897,A -85,B 0,C 180,E1 -8740.419,E2 -8740.419} C_VEL
LIN {X 0,Y 447.237,Z 430.838,A -85,B 0,C 180,E1 -8741.098,E2 -8741.098} C_VEL
LIN {X 0,Y 447.549,Z 422.499,A -85,B 0,C 180,E1 -8741.664,E2 -8741.664} C_VEL
LIN {X 0,Y 447.84,Z 414.005,A -85,B 0,C 180,E1 -8742.116,E2 -8742.116} C_VEL
LIN {X 0,Y 448.119,Z 404.743,A -85,B 0,C 180,E1 -8742.482,E2 -8742.482} C_VEL
LIN {X 0,Y 448.443,Z 393.782,A -85,B 0,C 180,E1 -8742.761,E2 -8742.761} C_VEL
LIN {X 0,Y 448.768,Z 338.067,A -85,B 0,C 180,E1 -8743.672,E2 -8743.672} C_VEL
LIN {X 0,Y 446.35,Z 319.771,A -85,B 0,C 180,E1 -8744.061,E2 -8744.061} C_VEL
LIN {X 0,Y 446.913,Z 303.994,A -85,B 0,C 180,E1 -8747.384,E2 -8747.384} C_VEL
LIN {X 0,Y 447.594,Z 287.369,A -85,B 0,C 180,E1 -8750.929,E2 -8750.929} C_VEL
LIN {X 0,Y 447.673,Z 281.751,A -85,B 0,C 180,E1 -8752.144,E2 -8752.144} C_VEL
LIN {X 0,Y 446.463,Z 274.687,A -85,B 0,C 180,E1 -8753.78,E2 -8753.78} C_VEL
LIN {X 0,Y 446.405,Z 274.692,A -85,B 0,C 180,E1 -8757.165,E2 -8757.165} C_VEL
LIN {X 0,Y 446.421,Z 274.69,A -85,B 0,C 180,E1 -8760.249,E2 -8760.249} C_VEL
LIN {X 0,Y 446.441,Z 274.685,A -85,B 0,C 180,E1 -8763.453,E2 -8763.453} C_VEL
LIN {X 0,Y 446.396,Z 274.695,A -85,B 0,C 180,E1 -8766.745,E2 -8766.745} C_VEL
LIN {X 0,Y 446.434,Z 274.687,A -85,B 0,C 180,E1 -8770.197,E2 -8770.197} C_VEL
LIN {X 0,Y 446.39,Z 274.696,A -85,B 0,C 180,E1 -8773.596,E2 -8773.596} C_VEL
LIN {X 0,Y 446.39,Z 274.69,A -85,B 0,C 180,E1 -8776.403,E2 -8776.403} C_VEL
LIN {X 0,Y 446.418,Z 274.688,A -85,B 0,C 180,E1 -8779.082,E2 -8779.082} C_VEL
LIN {X 0,Y 446.398,Z 274.686,A -85,B 0,C 180,E1 -8782.12,E2 -8782.12} C_VEL
LIN {X 0,Y 446.42,Z 274.691,A -85,B 0,C 180,E1 -8785.476,E2 -8785.476} C_VEL
LIN {X 0,Y 446.405,Z 274.686,A -85,B 0,C 180,E1 -8788.699,E2 -8788.699} C_VEL
LIN {X 0,Y 446.474,Z 274.681,A -85,B 0,C 180,E1 -8791.821,E2 -8791.821} C_VEL
LIN {X 0,Y 446.432,Z 274.683,A -85,B 0,C 180,E1 -8794.846,E2 -8794.846} C_VEL
LIN {X 0,Y 446.436,Z 274.682,A -85,B 0,C 180,E1 -8798.245,E2 -8798.245} C_VEL
LIN {X 0,Y 446.443,Z 274.683,A -85,B 0,C 180,E1 -8801.649,E2 -8801.649} C_VEL
LIN {X 0,Y 446.494,Z 274.675,A -85,B 0,C 180,E1 -8804.479,E2 -8804.479} C_VEL
LIN {X 0,Y 446.506,Z 274.678,A -85,B 0,C 180,E1 -8808.193,E2 -8808.193} C_VEL
LIN {X 0,Y 446.587,Z 274.659,A -85,B 0,C 180,E1 -8811.858,E2 -8811.858} C_VEL
LIN {X 0,Y 446.63,Z 274.664,A -85,B 0,C 180,E1 -8814.583,E2 -8814.583} C_VEL
LIN {X 0,Y 446.649,Z 274.653,A -85,B 0,C 180,E1 -8818.197,E2 -8818.197} C_VEL
LIN {X 0,Y 446.778,Z 274.639,A -85,B 0,C 180,E1 -8820,E2 -8820} C_VEL
LIN {X 0,Y 446.678,Z 274.65,A -85,B 0,C 180,E1 -8822.706,E2 -8822.706} C_VEL
LIN {X 0,Y 446.607,Z 274.661,A -85,B 0,C 180,E1 -8826.324,E2 -8826.324} C_VEL
LIN {X 0,Y 446.525,Z 274.674,A -85,B 0,C 180,E1 -8829.056,E2 -8829.056} C_VEL
LIN {X 0,Y 446.509,Z 274.67,A -85,B 0,C 180,E1 -8832.73,E2 -8832.73} C_VEL
LIN {X 0,Y 446.478,Z 274.675,A -85,B 0,C 180,E1 -8836.46,E2 -8836.46} C_VEL
LIN {X 0,Y 446.457,Z 274.686,A -85,B 0,C 180,E1 -8839.304,E2 -8839.304} C_VEL
LIN {X 0,Y 446.407,Z 274.691,A -85,B 0,C 180,E1 -8842.2,E2 -8842.2} C_VEL
LIN {X 0,Y 446.448,Z 274.684,A -85,B 0,C 180,E1 -8845.153,E2 -8845.153} C_VEL
LIN {X 0,Y 446.475,Z 274.683,A -85,B 0,C 180,E1 -8848.179,E2 -8848.179} C_VEL
LIN {X 0,Y 446.409,Z 274.687,A -85,B 0,C 180,E1 -8851.301,E2 -8851.301} C_VEL
LIN {X 0,Y 446.422,Z 274.687,A -85,B 0,C 180,E1 -8854.524,E2 -8854.524} C_VEL
LIN {X 0,Y 446.428,Z 274.691,A -85,B 0,C 180,E1 -8858.084,E2 -8858.084} C_VEL
LIN {X 0,Y 446.441,Z 274.689,A -85,B 0,C 180,E1 -8860.922,E2 -8860.922} C_VEL
LIN {X 0,Y 446.551,Z 274.743,A -85,B 0,C 180,E1 -8863.041,E2 -8863.041} C_VEL
LIN {X 0,Y 446.866,Z 279.203,A -85,B 0,C 180,E1 -8864.072,E2 -8864.072} C_VEL
LIN {X 0,Y 446.579,Z 292.76,A -85,B 0,C 180,E1 -8867.154,E2 -8867.154} C_VEL
LIN {X 0,Y 446.53,Z 296.5,A -85,B 0,C 180,E1 -8868.003,E2 -8868.003} C_VEL
LIN {X 0,Y 448.986,Z 311.231,A -85,B 0,C 180,E1 -8868.33,E2 -8868.33} C_VEL
LIN {X 0,Y 448.398,Z 372.929,A -85,B 0,C 180,E1 -8869.352,E2 -8869.352} C_VEL
LIN {X 0,Y 448.254,Z 382.59,A -85,B 0,C 180,E1 -8869.631,E2 -8869.631} C_VEL
LIN {X 0,Y 448.049,Z 392.781,A -85,B 0,C 180,E1 -8870.069,E2 -8870.069} C_VEL
LIN {X 0,Y 447.642,Z 402.93,A -85,B 0,C 180,E1 -8870.668,E2 -8870.668} C_VEL
LIN {X 0,Y 447.279,Z 412.041,A -85,B 0,C 180,E1 -8871.384,E2 -8871.384} C_VEL
LIN {X 0,Y 446.886,Z 420.071,A -85,B 0,C 180,E1 -8872.17,E2 -8872.17} C_VEL
LIN {X 0,Y 446.551,Z 426.942,A -85,B 0,C 180,E1 -8872.989,E2 -8872.989} C_VEL
LIN {X 0,Y 446.302,Z 432.686,A -85,B 0,C 180,E1 -8873.808,E2 -8873.808} C_VEL
LIN {X 0,Y 446.047,Z 438.09,A -85,B 0,C 180,E1 -8874.73,E2 -8874.73} C_VEL
LIN {X 0,Y 445.861,Z 442.793,A -85,B 0,C 180,E1 -8875.702,E2 -8875.702} C_VEL
LIN {X 0,Y 445.663,Z 446.733,A -85,B 0,C 180,E1 -8876.699,E2 -8876.699} C_VEL
LIN {X 0,Y 445.589,Z 449.561,A -85,B 0,C 180,E1 -8877.572,E2 -8877.572} C_VEL
LIN {X 0,Y 445.481,Z 452.189,A -85,B 0,C 180,E1 -8878.628,E2 -8878.628} C_VEL
LIN {X 0,Y 445.376,Z 454.046,A -85,B 0,C 180,E1 -8879.673,E2 -8879.673} C_VEL
LIN {X 0,Y 445.264,Z 455.182,A -85,B 0,C 180,E1 -8880.706,E2 -8880.706} C_VEL
LIN {X 0,Y 445.229,Z 455.713,A -85,B 0,C 180,E1 -8882.125,E2 -8882.125} C_VEL
LIN {X 0,Y 445.249,Z 454.706,A -85,B 0,C 180,E1 -8883.772,E2 -8883.772} C_VEL
LIN {X 0,Y 445.411,Z 452.401,A -85,B 0,C 180,E1 -8885.284,E2 -8885.284} C_VEL
LIN {X 0,Y 445.598,Z 448.568,A -85,B 0,C 180,E1 -8886.778,E2 -8886.778} C_VEL
LIN {X 0,Y 445.807,Z 443.527,A -85,B 0,C 180,E1 -8888.15,E2 -8888.15} C_VEL
LIN {X 0,Y 445.986,Z 438.413,A -85,B 0,C 180,E1 -8889.234,E2 -8889.234} C_VEL
LIN {X 0,Y 446.259,Z 432.739,A -85,B 0,C 180,E1 -8890.209,E2 -8890.209} C_VEL
LIN {X 0,Y 446.559,Z 426.403,A -85,B 0,C 180,E1 -8891.107,E2 -8891.107} C_VEL
LIN {X 0,Y 446.145,Z 422.239,A -85,B 0,C 180,E1 -8891.645,E2 -8891.645} C_VEL
LIN {X 0,Y 443.684,Z 415.108,A -85,B 0,C 180,E1 -8892.478,E2 -8892.478} C_VEL
LIN {X 0,Y 441.17,Z 407.361,A -85,B 0,C 180,E1 -8893.211,E2 -8893.211} C_VEL
LIN {X 0,Y 440.665,Z 402.23,A -85,B 0,C 180,E1 -8893.587,E2 -8893.587} C_VEL
LIN {X 0,Y 441.005,Z 392.455,A -85,B 0,C 180,E1 -8894.163,E2 -8894.163} C_VEL
LIN {X 0,Y 441.208,Z 382.744,A -85,B 0,C 180,E1 -8894.585,E2 -8894.585} C_VEL
LIN {X 0,Y 441.432,Z 373.469,A -85,B 0,C 180,E1 -8894.859,E2 -8894.859} C_VEL
LIN {X 0,Y 441.879,Z 311.634,A -85,B 0,C 180,E1 -8895.905,E2 -8895.905} C_VEL
LIN {X 0,Y 439.459,Z 296.989,A -85,B 0,C 180,E1 -8896.239,E2 -8896.239} C_VEL
LIN {X 0,Y 439.884,Z 284.444,A -85,B 0,C 180,E1 -8899.413,E2 -8899.413} C_VEL
LIN {X 0,Y 439.819,Z 277.244,A -85,B 0,C 180,E1 -8901.269,E2 -8901.269} C_VEL
LIN {X 0,Y 439.611,Z 275.541,A -85,B 0,C 180,E1 -8901.728,E2 -8901.728} C_VEL
LIN {X 0,Y 439.618,Z 275.533,A -85,B 0,C 180,E1 -8904.496,E2 -8904.496} C_VEL
LIN {X 0,Y 439.636,Z 275.533,A -85,B 0,C 180,E1 -8908.168,E2 -8908.168} C_VEL
LIN {X 0,Y 439.764,Z 275.521,A -85,B 0,C 180,E1 -8910,E2 -8910} C_VEL
LIN {X 0,Y 439.643,Z 275.529,A -85,B 0,C 180,E1 -8912.749,E2 -8912.749} C_VEL
LIN {X 0,Y 439.593,Z 275.539,A -85,B 0,C 180,E1 -8916.425,E2 -8916.425} C_VEL
LIN {X 0,Y 439.5,Z 275.546,A -85,B 0,C 180,E1 -8919.201,E2 -8919.201} C_VEL
LIN {X 0,Y 439.467,Z 275.552,A -85,B 0,C 180,E1 -8922.937,E2 -8922.937} C_VEL
LIN {X 0,Y 439.447,Z 275.559,A -85,B 0,C 180,E1 -8926.348,E2 -8926.348} C_VEL
LIN {X 0,Y 439.402,Z 275.558,A -85,B 0,C 180,E1 -8929.626,E2 -8929.626} C_VEL
LIN {X 0,Y 439.364,Z 275.57,A -85,B 0,C 180,E1 -8932.575,E2 -8932.575} C_VEL
LIN {X 0,Y 439.399,Z 275.559,A -85,B 0,C 180,E1 -8935.584,E2 -8935.584} C_VEL
LIN {X 0,Y 439.416,Z 275.562,A -85,B 0,C 180,E1 -8938.673,E2 -8938.673} C_VEL
LIN {X 0,Y 439.366,Z 275.563,A -85,B 0,C 180,E1 -8942.029,E2 -8942.029} C_VEL
LIN {X 0,Y 439.388,Z 275.566,A -85,B 0,C 180,E1 -8945.339,E2 -8945.339} C_VEL
LIN {X 0,Y 439.379,Z 275.562,A -85,B 0,C 180,E1 -8948.594,E2 -8948.594} C_VEL
LIN {X 0,Y 439.383,Z 275.568,A -85,B 0,C 180,E1 -8951.256,E2 -8951.256} C_VEL
LIN {X 0,Y 439.397,Z 275.56,A -85,B 0,C 180,E1 -8954.728,E2 -8954.728} C_VEL
LIN {X 0,Y 439.406,Z 275.564,A -85,B 0,C 180,E1 -8957.797,E2 -8957.797} C_VEL
LIN {X 0,Y 439.442,Z 275.555,A -85,B 0,C 180,E1 -8960.229,E2 -8960.229} C_VEL
LIN {X 0,Y 439.369,Z 275.57,A -85,B 0,C 180,E1 -8963.712,E2 -8963.712} C_VEL
LIN {X 0,Y 439.364,Z 275.563,A -85,B 0,C 180,E1 -8967.053,E2 -8967.053} C_VEL
LIN {X 0,Y 439.387,Z 275.566,A -85,B 0,C 180,E1 -8970.274,E2 -8970.274} C_VEL
LIN {X 0,Y 439.424,Z 275.557,A -85,B 0,C 180,E1 -8973.588,E2 -8973.588} C_VEL
LIN {X 0,Y 439.377,Z 275.568,A -85,B 0,C 180,E1 -8976.429,E2 -8976.429} C_VEL
LIN {X 0,Y 439.376,Z 275.562,A -85,B 0,C 180,E1 -8979.396,E2 -8979.396} C_VEL
LIN {X 0,Y 439.419,Z 275.562,A -85,B 0,C 180,E1 -8982.309,E2 -8982.309} C_VEL
LIN {X 0,Y 439.436,Z 275.556,A -85,B 0,C 180,E1 -8985.173,E2 -8985.173} C_VEL
LIN {X 0,Y 439.471,Z 275.551,A -85,B 0,C 180,E1 -8988.001,E2 -8988.001} C_VEL
LIN {X 0,Y 439.536,Z 275.542,A -85,B 0,C 180,E1 -8991.726,E2 -8991.726} C_VEL
LIN {X 0,Y 439.604,Z 275.536,A -85,B 0,C 180,E1 -8994.495,E2 -8994.495} C_VEL
LIN {X 0,Y 439.623,Z 275.531,A -85,B 0,C 180,E1 -8998.168,E2 -8998.168} C_VEL
LIN {X 0,Y 439.749,Z 275.515,A -85,B 0,C 180,E1 -9000,E2 -9000} C_VEL
LIN {X 0,Y 439.628,Z 275.533,A -85,B 0,C 180,E1 -9002.749,E2 -9002.749} C_VEL
LIN {X 0,Y 439.602,Z 275.534,A -85,B 0,C 180,E1 -9006.425,E2 -9006.425} C_VEL
LIN {X 0,Y 439.489,Z 275.553,A -85,B 0,C 180,E1 -9009.202,E2 -9009.202} C_VEL
LIN {X 0,Y 439.492,Z 275.547,A -85,B 0,C 180,E1 -9012.727,E2 -9012.727} C_VEL
LIN {X 0,Y 439.435,Z 275.555,A -85,B 0,C 180,E1 -9016.349,E2 -9016.349} C_VEL
LIN {X 0,Y 439.391,Z 275.566,A -85,B 0,C 180,E1 -9019.627,E2 -9019.627} C_VEL
LIN {X 0,Y 439.353,Z 275.565,A -85,B 0,C 180,E1 -9022.576,E2 -9022.576} C_VEL
LIN {X 0,Y 439.394,Z 275.562,A -85,B 0,C 180,E1 -9025.585,E2 -9025.585} C_VEL
LIN {X 0,Y 439.406,Z 275.56,A -85,B 0,C 180,E1 -9028.674,E2 -9028.674} C_VEL
LIN {X 0,Y 439.359,Z 275.569,A -85,B 0,C 180,E1 -9032.031,E2 -9032.031} C_VEL
LIN {X 0,Y 439.386,Z 275.56,A -85,B 0,C 180,E1 -9035.341,E2 -9035.341} C_VEL
LIN {X 0,Y 439.361,Z 275.57,A -85,B 0,C 180,E1 -9038.597,E2 -9038.597} C_VEL
LIN {X 0,Y 439.38,Z 275.562,A -85,B 0,C 180,E1 -9041.257,E2 -9041.257} C_VEL
LIN {X 0,Y 439.391,Z 275.568,A -85,B 0,C 180,E1 -9044.73,E2 -9044.73} C_VEL
LIN {X 0,Y 439.377,Z 275.562,A -85,B 0,C 180,E1 -9047.795,E2 -9047.795} C_VEL
LIN {X 0,Y 439.388,Z 275.561,A -85,B 0,C 180,E1 -9050.225,E2 -9050.225} C_VEL
LIN {X 0,Y 439.368,Z 275.563,A -85,B 0,C 180,E1 -9053.714,E2 -9053.714} C_VEL
LIN {X 0,Y 439.368,Z 275.57,A -85,B 0,C 180,E1 -9057.055,E2 -9057.055} C_VEL
LIN {X 0,Y 439.372,Z 275.562,A -85,B 0,C 180,E1 -9060.274,E2 -9060.274} C_VEL
LIN {X 0,Y 439.376,Z 275.57,A -85,B 0,C 180,E1 -9063.394,E2 -9063.394} C_VEL
LIN {X 0,Y 439.458,Z 275.654,A -85,B 0,C 180,E1 -9065.881,E2 -9065.881} C_VEL
LIN {X 0,Y 440.74,Z 283.109,A -85,B 0,C 180,E1 -9067.648,E2 -9067.648} C_VEL
LIN {X 0,Y 440.679,Z 290.066,A -85,B 0,C 180,E1 -9069.217,E2 -9069.217} C_VEL
LIN {X 0,Y 439.876,Z 307.419,A -85,B 0,C 180,E1 -9073.048,E2 -9073.048} C_VEL
LIN {X 0,Y 439.33,Z 320.027,A -85,B 0,C 180,E1 -9075.797,E2 -9075.797} C_VEL
LIN {X 0,Y 441.813,Z 339.188,A -85,B 0,C 180,E1 -9076.196,E2 -9076.196} C_VEL
LIN {X 0,Y 441.348,Z 397.317,A -85,B 0,C 180,E1 -9077.177,E2 -9077.177} C_VEL
LIN {X 0,Y 441.034,Z 407.807,A -85,B 0,C 180,E1 -9077.49,E2 -9077.49} C_VEL
LIN {X 0,Y 440.652,Z 419.546,A -85,B 0,C 180,E1 -9078.034,E2 -9078.034} C_VEL
LIN {X 0,Y 440.257,Z 428.468,A -85,B 0,C 180,E1 -9078.607,E2 -9078.607} C_VEL
LIN {X 0,Y 439.913,Z 436.949,A -85,B 0,C 180,E1 -9079.297,E2 -9079.297} C_VEL
LIN {X 0,Y 439.546,Z 444.95,A -85,B 0,C 180,E1 -9080.103,E2 -9080.103} C_VEL
LIN {X 0,Y 439.275,Z 450.704,A -85,B 0,C 180,E1 -9080.794,E2 -9080.794} C_VEL
LIN {X 0,Y 438.917,Z 457.126,A -85,B 0,C 180,E1 -9081.715,E2 -9081.715} C_VEL
LIN {X 0,Y 438.716,Z 462.466,A -85,B 0,C 180,E1 -9082.637,E2 -9082.637} C_VEL
LIN {X 0,Y 438.52,Z 467.963,A -85,B 0,C 180,E1 -9083.809,E2 -9083.809} C_VEL
LIN {X 0,Y 438.449,Z 472.155,A -85,B 0,C 180,E1 -9084.942,E2 -9084.942} C_VEL
LIN {X 0,Y 438.32,Z 474.841,A -85,B 0,C 180,E1 -9085.862,E2 -9085.862} C_VEL
LIN {X 0,Y 438.35,Z 477.783,A -85,B 0,C 180,E1 -9087.243,E2 -9087.243} C_VEL
LIN {X 0,Y 438.277,Z 479.06,A -85,B 0,C 180,E1 -9088.162,E2 -9088.162} C_VEL
LIN {X 0,Y 438.25,Z 479.86,A -85,B 0,C 180,E1 -9089.081,E2 -9089.081} C_VEL
LIN {X 0,Y 438.252,Z 480.159,A -85,B 0,C 180,E1 -9090,E2 -9090} C_VEL
LIN {X 0,Y 438.25,Z 479.866,A -85,B 0,C 180,E1 -9090.919,E2 -9090.919} C_VEL
LIN {X 0,Y 438.277,Z 479.092,A -85,B 0,C 180,E1 -9091.838,E2 -9091.838} C_VEL
LIN {X 0,Y 438.35,Z 477.843,A -85,B 0,C 180,E1 -9092.757,E2 -9092.757} C_VEL
LIN {X 0,Y 438.32,Z 474.928,A -85,B 0,C 180,E1 -9094.138,E2 -9094.138} C_VEL
LIN {X 0,Y 438.448,Z 472.279,A -85,B 0,C 180,E1 -9095.058,E2 -9095.058} C_VEL
LIN {X 0,Y 438.496,Z 468.256,A -85,B 0,C 180,E1 -9096.16,E2 -9096.16} C_VEL
LIN {X 0,Y 438.708,Z 463.863,A -85,B 0,C 180,E1 -9097.131,E2 -9097.131} C_VEL
LIN {X 0,Y 438.873,Z 458.832,A -85,B 0,C 180,E1 -9098.055,E2 -9098.055} C_VEL
LIN {X 0,Y 439.173,Z 452.779,A -85,B 0,C 180,E1 -9098.976,E2 -9098.976} C_VEL
LIN {X 0,Y 439.582,Z 445.416,A -85,B 0,C 180,E1 -9099.896,E2 -9099.896} C_VEL
LIN {X 0,Y 439.944,Z 437.538,A -85,B 0,C 180,E1 -9100.702,E2 -9100.702} C_VEL
LIN {X 0,Y 440.332,Z 429.226,A -85,B 0,C 180,E1 -9101.391,E2 -9101.391} C_VEL
LIN {X 0,Y 440.757,Z 418.643,A -85,B 0,C 180,E1 -9102.08,E2 -9102.08} C_VEL
LIN {X 0,Y 441.114,Z 407.233,A -85,B 0,C 180,E1 -9102.596,E2 -9102.596} C_VEL
LIN {X 0,Y 441.47,Z 397.065,A -85,B 0,C 180,E1 -9102.895,E2 -9102.895} C_VEL
LIN {X 0,Y 441.864,Z 338.542,A -85,B 0,C 180,E1 -9103.887,E2 -9103.887} C_VEL
LIN {X 0,Y 439.353,Z 319.526,A -85,B 0,C 180,E1 -9104.308,E2 -9104.308} C_VEL
LIN {X 0,Y 439.916,Z 303.835,A -85,B 0,C 180,E1 -9107.67,E2 -9107.67} C_VEL
LIN {X 0,Y 440.696,Z 287.195,A -85,B 0,C 180,E1 -9111.272,E2 -9111.272} C_VEL
LIN {X 0,Y 440.639,Z 282.457,A -85,B 0,C 180,E1 -9112.321,E2 -9112.321} C_VEL
LIN {X 0,Y 439.407,Z 275.566,A -85,B 0,C 180,E1 -9113.974,E2 -9113.974} C_VEL
LIN {X 0,Y 439.366,Z 275.572,A -85,B 0,C 180,E1 -9116.607,E2 -9116.607} C_VEL
LIN {X 0,Y 439.367,Z 275.567,A -85,B 0,C 180,E1 -9119.726,E2 -9119.726} C_VEL
LIN {X 0,Y 439.367,Z 275.571,A -85,B 0,C 180,E1 -9122.945,E2 -9122.945} C_VEL
LIN {X 0,Y 439.368,Z 275.566,A -85,B 0,C 180,E1 -9126.286,E2 -9126.286} C_VEL
LIN {X 0,Y 439.396,Z 275.565,A -85,B 0,C 180,E1 -9129.848,E2 -9129.848} C_VEL
LIN {X 0,Y 439.363,Z 275.567,A -85,B 0,C 180,E1 -9132.624,E2 -9132.624} C_VEL
LIN {X 0,Y 439.391,Z 275.567,A -85,B 0,C 180,E1 -9135.27,E2 -9135.27} C_VEL
LIN {X 0,Y 439.38,Z 275.562,A -85,B 0,C 180,E1 -9138.743,E2 -9138.743} C_VEL
LIN {X 0,Y 439.36,Z 275.569,A -85,B 0,C 180,E1 -9141.608,E2 -9141.608} C_VEL
LIN {X 0,Y 439.39,Z 275.561,A -85,B 0,C 180,E1 -9144.843,E2 -9144.843} C_VEL
LIN {X 0,Y 439.362,Z 275.567,A -85,B 0,C 180,E1 -9148.139,E2 -9148.139} C_VEL
LIN {X 0,Y 439.422,Z 275.56,A -85,B 0,C 180,E1 -9151.598,E2 -9151.598} C_VEL
LIN {X 0,Y 439.386,Z 275.564,A -85,B 0,C 180,E1 -9154.414,E2 -9154.414} C_VEL
LIN {X 0,Y 439.352,Z 275.563,A -85,B 0,C 180,E1 -9157.424,E2 -9157.424} C_VEL
LIN {X 0,Y 439.429,Z 275.559,A -85,B 0,C 180,E1 -9160.663,E2 -9160.663} C_VEL
LIN {X 0,Y 439.449,Z 275.552,A -85,B 0,C 180,E1 -9164.224,E2 -9164.224} C_VEL
LIN {X 0,Y 439.472,Z 275.553,A -85,B 0,C 180,E1 -9168.001,E2 -9168.001} C_VEL
LIN {X 0,Y 439.535,Z 275.538,A -85,B 0,C 180,E1 -9171.726,E2 -9171.726} C_VEL
LIN {X 0,Y 439.605,Z 275.538,A -85,B 0,C 180,E1 -9174.496,E2 -9174.496} C_VEL
LIN {X 0,Y 439.62,Z 275.529,A -85,B 0,C 180,E1 -9178.168,E2 -9178.168} C_VEL
LIN {X 0,Y 439.749,Z 275.515,A -85,B 0,C 180,E1 -9180,E2 -9180} C_VEL
LIN {X 0,Y 439.628,Z 275.528,A -85,B 0,C 180,E1 -9182.749,E2 -9182.749} C_VEL
LIN {X 0,Y 439.569,Z 275.537,A -85,B 0,C 180,E1 -9186.509,E2 -9186.509} C_VEL
LIN {X 0,Y 439.487,Z 275.552,A -85,B 0,C 180,E1 -9189.202,E2 -9189.202} C_VEL
LIN {X 0,Y 439.453,Z 275.551,A -85,B 0,C 180,E1 -9192.938,E2 -9192.938} C_VEL
LIN {X 0,Y 439.435,Z 275.553,A -85,B 0,C 180,E1 -9196.349,E2 -9196.349} C_VEL
LIN {X 0,Y 439.391,Z 275.568,A -85,B 0,C 180,E1 -9199.627,E2 -9199.627} C_VEL
LIN {X 0,Y 439.354,Z 275.568,A -85,B 0,C 180,E1 -9202.576,E2 -9202.576} C_VEL
LIN {X 0,Y 439.396,Z 275.567,A -85,B 0,C 180,E1 -9205.586,E2 -9205.586} C_VEL
LIN {X 0,Y 439.416,Z 275.558,A -85,B 0,C 180,E1 -9208.674,E2 -9208.674} C_VEL
LIN {X 0,Y 439.365,Z 275.57,A -85,B 0,C 180,E1 -9211.861,E2 -9211.861} C_VEL
LIN {X 0,Y 439.393,Z 275.559,A -85,B 0,C 180,E1 -9215.157,E2 -9215.157} C_VEL
LIN {X 0,Y 439.388,Z 275.567,A -85,B 0,C 180,E1 -9218.595,E2 -9218.595} C_VEL
LIN {X 0,Y 439.398,Z 275.565,A -85,B 0,C 180,E1 -9221.26,E2 -9221.26} C_VEL
LIN {X 0,Y 439.492,Z 275.605,A -85,B 0,C 180,E1 -9222.887,E2 -9222.887} C_VEL
LIN {X 0,Y 439.904,Z 279.062,A -85,B 0,C 180,E1 -9223.711,E2 -9223.711} C_VEL
LIN {X 0,Y 439.574,Z 293.37,A -85,B 0,C 180,E1 -9227.004,E2 -9227.004} C_VEL
LIN {X 0,Y 439.518,Z 296.67,A -85,B 0,C 180,E1 -9227.763,E2 -9227.763} C_VEL
LIN {X 0,Y 442.098,Z 312.064,A -85,B 0,C 180,E1 -9228.114,E2 -9228.114} C_VEL
LIN {X 0,Y 441.51,Z 373.569,A -85,B 0,C 180,E1 -9229.153,E2 -9229.153} C_VEL
LIN {X 0,Y 441.334,Z 383.593,A -85,B 0,C 180,E1 -9229.455,E2 -9229.455} C_VEL
LIN {X 0,Y 441.049,Z 395.385,A -85,B 0,C 180,E1 -9229.998,E2 -9229.998} C_VEL
LIN {X 0,Y 440.612,Z 405.411,A -85,B 0,C 180,E1 -9230.653,E2 -9230.653} C_VEL
LIN {X 0,Y 440.229,Z 413.91,A -85,B 0,C 180,E1 -9231.363,E2 -9231.363} C_VEL
LIN {X 0,Y 439.899,Z 420.607,A -85,B 0,C 180,E1 -9232.043,E2 -9232.043} C_VEL
LIN {X 0,Y 439.541,Z 427.484,A -85,B 0,C 180,E1 -9232.882,E2 -9232.882} C_VEL
LIN {X 0,Y 439.262,Z 433.107,A -85,B 0,C 180,E1 -9233.703,E2 -9233.703} C_VEL
LIN {X 0,Y 438.977,Z 438.963,A -85,B 0,C 180,E1 -9234.737,E2 -9234.737} C_VEL
LIN {X 0,Y 438.759,Z 444.276,A -85,B 0,C 180,E1 -9235.902,E2 -9235.902} C_VEL
LIN {X 0,Y 438.535,Z 448.177,A -85,B 0,C 180,E1 -9236.984,E2 -9236.984} C_VEL
LIN {X 0,Y 438.461,Z 451.426,A -85,B 0,C 180,E1 -9238.16,E2 -9238.16} C_VEL
LIN {X 0,Y 438.335,Z 453.393,A -85,B 0,C 180,E1 -9239.133,E2 -9239.133} C_VEL
LIN {X 0,Y 438.213,Z 454.871,A -85,B 0,C 180,E1 -9240.188,E2 -9240.188} C_VEL
LIN {X 0,Y 438.13,Z 455.911,A -85,B 0,C 180,E1 -9241.915,E2 -9241.915} C_VEL
LIN {X 0,Y 438.135,Z 455.406,A -85,B 0,C 180,E1 -9243.312,E2 -9243.312} C_VEL
LIN {X 0,Y 438.224,Z 454.303,A -85,B 0,C 180,E1 -9244.342,E2 -9244.342} C_VEL
LIN {X 0,Y 438.335,Z 452.533,A -85,B 0,C 180,E1 -9245.364,E2 -9245.364} C_VEL
LIN {X 0,Y 438.541,Z 448.642,A -85,B 0,C 180,E1 -9246.882,E2 -9246.882} C_VEL
LIN {X 0,Y 438.759,Z 443.528,A -85,B 0,C 180,E1 -9248.286,E2 -9248.286} C_VEL
LIN {X 0,Y 438.944,Z 438.425,A -85,B 0,C 180,E1 -9249.376,E2 -9249.376} C_VEL
LIN {X 0,Y 439.315,Z 431.378,A -85,B 0,C 180,E1 -9250.582,E2 -9250.582} C_VEL
LIN {X 0,Y 439.694,Z 422.767,A -85,B 0,C 180,E1 -9251.719,E2 -9251.719} C_VEL
LIN {X 0,Y 440.13,Z 414.585,A -85,B 0,C 180,E1 -9252.579,E2 -9252.579} C_VEL
LIN {X 0,Y 440.446,Z 407.209,A -85,B 0,C 180,E1 -9253.215,E2 -9253.215} C_VEL
LIN {X 0,Y 440.665,Z 402.23,A -85,B 0,C 180,E1 -9253.587,E2 -9253.587} C_VEL
LIN {X 0,Y 440.322,Z 396.951,A -85,B 0,C 180,E1 -9253.934,E2 -9253.934} C_VEL
LIN {X 0,Y 438.958,Z 391.728,A -85,B 0,C 180,E1 -9254.259,E2 -9254.259} C_VEL
LIN {X 0,Y 435.383,Z 380.199,A -85,B 0,C 180,E1 -9254.847,E2 -9254.847} C_VEL
LIN {X 0,Y 434.496,Z 373.575,A -85,B 0,C 180,E1 -9255.058,E2 -9255.058} C_VEL
LIN {X 0,Y 434.839,Z 311.167,A -85,B 0,C 180,E1 -9256.134,E2 -9256.134} C_VEL
LIN {X 0,Y 432.464,Z 297.132,A -85,B 0,C 180,E1 -9256.473,E2 -9256.473} C_VEL
LIN {X 0,Y 432.909,Z 284.508,A -85,B 0,C 180,E1 -9259.713,E2 -9259.713} C_VEL
LIN {X 0,Y 432.704,Z 277.338,A -85,B 0,C 180,E1 -9261.595,E2 -9261.595} C_VEL
LIN {X 0,Y 432.576,Z 276.417,A -85,B 0,C 180,E1 -9261.851,E2 -9261.851} C_VEL
LIN {X 0,Y 432.595,Z 276.409,A -85,B 0,C 180,E1 -9264.406,E2 -9264.406} C_VEL
LIN {X 0,Y 432.605,Z 276.41,A -85,B 0,C 180,E1 -9268.138,E2 -9268.138} C_VEL
LIN {X 0,Y 432.734,Z 276.396,A -85,B 0,C 180,E1 -9270,E2 -9270} C_VEL
LIN {X 0,Y 432.594,Z 276.407,A -85,B 0,C 180,E1 -9272.794,E2 -9272.794} C_VEL
LIN {X 0,Y 432.587,Z 276.409,A -85,B 0,C 180,E1 -9275.594,E2 -9275.594} C_VEL
LIN {X 0,Y 432.484,Z 276.426,A -85,B 0,C 180,E1 -9278.41,E2 -9278.41} C_VEL
LIN {X 0,Y 432.46,Z 276.43,A -85,B 0,C 180,E1 -9282.196,E2 -9282.196} C_VEL
LIN {X 0,Y 432.431,Z 276.43,A -85,B 0,C 180,E1 -9286.038,E2 -9286.038} C_VEL
LIN {X 0,Y 432.387,Z 276.432,A -85,B 0,C 180,E1 -9289.484,E2 -9289.484} C_VEL
LIN {X 0,Y 432.318,Z 276.446,A -85,B 0,C 180,E1 -9292.964,E2 -9292.964} C_VEL
LIN {X 0,Y 432.361,Z 276.436,A -85,B 0,C 180,E1 -9296.032,E2 -9296.032} C_VEL
LIN {X 0,Y 432.341,Z 276.443,A -85,B 0,C 180,E1 -9299.187,E2 -9299.187} C_VEL
LIN {X 0,Y 432.32,Z 276.442,A -85,B 0,C 180,E1 -9302.442,E2 -9302.442} C_VEL
LIN {X 0,Y 432.339,Z 276.441,A -85,B 0,C 180,E1 -9305.631,E2 -9305.631} C_VEL
LIN {X 0,Y 432.346,Z 276.446,A -85,B 0,C 180,E1 -9309.342,E2 -9309.342} C_VEL
LIN {X 0,Y 432.328,Z 276.443,A -85,B 0,C 180,E1 -9311.796,E2 -9311.796} C_VEL
LIN {X 0,Y 432.373,Z 276.441,A -85,B 0,C 180,E1 -9315.658,E2 -9315.658} C_VEL
LIN {X 0,Y 432.367,Z 276.435,A -85,B 0,C 180,E1 -9318.391,E2 -9318.391} C_VEL
LIN {X 0,Y 432.344,Z 276.445,A -85,B 0,C 180,E1 -9321.851,E2 -9321.851} C_VEL
LIN {X 0,Y 432.333,Z 276.441,A -85,B 0,C 180,E1 -9325.322,E2 -9325.322} C_VEL
LIN {X 0,Y 432.314,Z 276.442,A -85,B 0,C 180,E1 -9328.653,E2 -9328.653} C_VEL
LIN {X 0,Y 432.372,Z 276.435,A -85,B 0,C 180,E1 -9331.368,E2 -9331.368} C_VEL
LIN {X 0,Y 432.355,Z 276.442,A -85,B 0,C 180,E1 -9333.967,E2 -9333.967} C_VEL
LIN {X 0,Y 432.309,Z 276.443,A -85,B 0,C 180,E1 -9337.035,E2 -9337.035} C_VEL
LIN {X 0,Y 432.376,Z 276.441,A -85,B 0,C 180,E1 -9340.514,E2 -9340.514} C_VEL
LIN {X 0,Y 432.419,Z 276.43,A -85,B 0,C 180,E1 -9343.961,E2 -9343.961} C_VEL
LIN {X 0,Y 432.447,Z 276.425,A -85,B 0,C 180,E1 -9347.803,E2 -9347.803} C_VEL
LIN {X 0,Y 432.48,Z 276.421,A -85,B 0,C 180,E1 -9351.59,E2 -9351.59} C_VEL
LIN {X 0,Y 432.581,Z 276.41,A -85,B 0,C 180,E1 -9354.406,E2 -9354.406} C_VEL
LIN {X 0,Y 432.593,Z 276.407,A -85,B 0,C 180,E1 -9358.138,E2 -9358.138} C_VEL
LIN {X 0,Y 432.719,Z 276.391,A -85,B 0,C 180,E1 -9360,E2 -9360} C_VEL
LIN {X 0,Y 432.58,Z 276.411,A -85,B 0,C 180,E1 -9362.794,E2 -9362.794} C_VEL
LIN {X 0,Y 432.557,Z 276.411,A -85,B 0,C 180,E1 -9366.53,E2 -9366.53} C_VEL
LIN {X 0,Y 432.433,Z 276.434,A -85,B 0,C 180,E1 -9369.353,E2 -9369.353} C_VEL
LIN {X 0,Y 432.433,Z 276.427,A -85,B 0,C 180,E1 -9372.812,E2 -9372.812} C_VEL
LIN {X 0,Y 432.401,Z 276.431,A -85,B 0,C 180,E1 -9376.479,E2 -9376.479} C_VEL
LIN {X 0,Y 432.327,Z 276.446,A -85,B 0,C 180,E1 -9379.961,E2 -9379.961} C_VEL
LIN {X 0,Y 432.308,Z 276.442,A -85,B 0,C 180,E1 -9382.965,E2 -9382.965} C_VEL
LIN {X 0,Y 432.354,Z 276.445,A -85,B 0,C 180,E1 -9386.033,E2 -9386.033} C_VEL
LIN {X 0,Y 432.332,Z 276.439,A -85,B 0,C 180,E1 -9389.188,E2 -9389.188} C_VEL
LIN {X 0,Y 432.313,Z 276.447,A -85,B 0,C 180,E1 -9392.444,E2 -9392.444} C_VEL
LIN {X 0,Y 432.336,Z 276.439,A -85,B 0,C 180,E1 -9395.633,E2 -9395.633} C_VEL
LIN {X 0,Y 432.325,Z 276.445,A -85,B 0,C 180,E1 -9398.714,E2 -9398.714} C_VEL
LIN {X 0,Y 432.325,Z 276.44,A -85,B 0,C 180,E1 -9401.798,E2 -9401.798} C_VEL
LIN {X 0,Y 432.326,Z 276.444,A -85,B 0,C 180,E1 -9404.348,E2 -9404.348} C_VEL
LIN {X 0,Y 432.309,Z 276.447,A -85,B 0,C 180,E1 -9407.017,E2 -9407.017} C_VEL
LIN {X 0,Y 432.325,Z 276.44,A -85,B 0,C 180,E1 -9409.822,E2 -9409.822} C_VEL
LIN {X 0,Y 432.301,Z 276.451,A -85,B 0,C 180,E1 -9413.023,E2 -9413.023} C_VEL
LIN {X 0,Y 432.353,Z 276.437,A -85,B 0,C 180,E1 -9415.998,E2 -9415.998} C_VEL
LIN {X 0,Y 432.342,Z 276.443,A -85,B 0,C 180,E1 -9419.491,E2 -9419.491} C_VEL
LIN {X 0,Y 432.339,Z 276.442,A -85,B 0,C 180,E1 -9421.875,E2 -9421.875} C_VEL
LIN {X 0,Y 432.394,Z 276.438,A -85,B 0,C 180,E1 -9425.643,E2 -9425.643} C_VEL
LIN {X 0,Y 433.025,Z 280.029,A -85,B 0,C 180,E1 -9426.57,E2 -9426.57} C_VEL
LIN {X 0,Y 433.818,Z 285.186,A -85,B 0,C 180,E1 -9427.802,E2 -9427.802} C_VEL
LIN {X 0,Y 433.561,Z 293.098,A -85,B 0,C 180,E1 -9429.604,E2 -9429.604} C_VEL
LIN {X 0,Y 432.849,Z 308.27,A -85,B 0,C 180,E1 -9433.007,E2 -9433.007} C_VEL
LIN {X 0,Y 432.319,Z 319.796,A -85,B 0,C 180,E1 -9435.562,E2 -9435.562} C_VEL
LIN {X 0,Y 434.899,Z 340.065,A -85,B 0,C 180,E1 -9436.001,E2 -9436.001} C_VEL
LIN {X 0,Y 434.434,Z 396.627,A -85,B 0,C 180,E1 -9436.97,E2 -9436.97} C_VEL
LIN {X 0,Y 434.106,Z 406.46,A -85,B 0,C 180,E1 -9437.257,E2 -9437.257} C_VEL
LIN {X 0,Y 433.739,Z 418.164,A -85,B 0,C 180,E1 -9437.781,E2 -9437.781} C_VEL
LIN {X 0,Y 433.288,Z 428.128,A -85,B 0,C 180,E1 -9438.421,E2 -9438.421} C_VEL
LIN {X 0,Y 432.928,Z 436.635,A -85,B 0,C 180,E1 -9439.122,E2 -9439.122} C_VEL
LIN {X 0,Y 432.542,Z 444.656,A -85,B 0,C 180,E1 -9439.941,E2 -9439.941} C_VEL
LIN {X 0,Y 432.239,Z 450.426,A -85,B 0,C 180,E1 -9440.643,E2 -9440.643} C_VEL
LIN {X 0,Y 431.867,Z 456.863,A -85,B 0,C 180,E1 -9441.578,E2 -9441.578} C_VEL
LIN {X 0,Y 431.645,Z 462.216,A -85,B 0,C 180,E1 -9442.516,E2 -9442.516} C_VEL
LIN {X 0,Y 431.499,Z 466.782,A -85,B 0,C 180,E1 -9443.478,E2 -9443.478} C_VEL
LIN {X 0,Y 431.377,Z 470.396,A -85,B 0,C 180,E1 -9444.39,E2 -9444.39} C_VEL
LIN {X 0,Y 431.3,Z 473.428,A -85,B 0,C 180,E1 -9445.327,E2 -9445.327} C_VEL
LIN {X 0,Y 431.217,Z 475.778,A -85,B 0,C 180,E1 -9446.262,E2 -9446.262} C_VEL
LIN {X 0,Y 431.246,Z 477.569,A -85,B 0,C 180,E1 -9447.198,E2 -9447.198} C_VEL
LIN {X 0,Y 431.202,Z 478.855,A -85,B 0,C 180,E1 -9448.132,E2 -9448.132} C_VEL
LIN {X 0,Y 431.166,Z 479.661,A -85,B 0,C 180,E1 -9449.066,E2 -9449.066} C_VEL
LIN {X 0,Y 431.166,Z 479.962,A -85,B 0,C 180,E1 -9450,E2 -9450} C_VEL
LIN {X 0,Y 431.166,Z 479.672,A -85,B 0,C 180,E1 -9450.934,E2 -9450.934} C_VEL
LIN {X 0,Y 431.202,Z 478.905,A -85,B 0,C 180,E1 -9451.868,E2 -9451.868} C_VEL
LIN {X 0,Y 431.246,Z 477.66,A -85,B 0,C 180,E1 -9452.802,E2 -9452.802} C_VEL
LIN {X 0,Y 431.238,Z 474.75,A -85,B 0,C 180,E1 -9454.206,E2 -9454.206} C_VEL
LIN {X 0,Y 431.362,Z 472.107,A -85,B 0,C 180,E1 -9455.141,E2 -9455.141} C_VEL
LIN {X 0,Y 431.482,Z 466.914,A -85,B 0,C 180,E1 -9456.547,E2 -9456.547} C_VEL
LIN {X 0,Y 431.693,Z 461.334,A -85,B 0,C 180,E1 -9457.718,E2 -9457.718} C_VEL
LIN {X 0,Y 432.063,Z 454.331,A -85,B 0,C 180,E1 -9458.889,E2 -9458.889} C_VEL
LIN {X 0,Y 432.525,Z 446.305,A -85,B 0,C 180,E1 -9459.941,E2 -9459.941} C_VEL
LIN {X 0,Y 432.91,Z 438.648,A -85,B 0,C 180,E1 -9460.76,E2 -9460.76} C_VEL
LIN {X 0,Y 433.294,Z 430.621,A -85,B 0,C 180,E1 -9461.46,E2 -9461.46} C_VEL
LIN {X 0,Y 433.637,Z 422.326,A -85,B 0,C 180,E1 -9462.044,E2 -9462.044} C_VEL
LIN {X 0,Y 433.974,Z 413.901,A -85,B 0,C 180,E1 -9462.509,E2 -9462.509} C_VEL
LIN {X 0,Y 434.297,Z 404.754,A -85,B 0,C 180,E1 -9462.886,E2 -9462.886} C_VEL
LIN {X 0,Y 434.644,Z 395.001,A -85,B 0,C 180,E1 -9463.151,E2 -9463.151} C_VEL
LIN {X 0,Y 434.954,Z 338.7,A -85,B 0,C 180,E1 -9464.115,E2 -9464.115} C_VEL
LIN {X 0,Y 432.323,Z 319.369,A -85,B 0,C 180,E1 -9464.546,E2 -9464.546} C_VEL
LIN {X 0,Y 432.914,Z 304.789,A -85,B 0,C 180,E1 -9467.721,E2 -9467.721} C_VEL
LIN {X 0,Y 433.726,Z 288.133,A -85,B 0,C 180,E1 -9471.381,E2 -9471.381} C_VEL
LIN {X 0,Y 433.596,Z 283.189,A -85,B 0,C 180,E1 -9472.498,E2 -9472.498} C_VEL
LIN {X 0,Y 432.371,Z 276.442,A -85,B 0,C 180,E1 -9474.097,E2 -9474.097} C_VEL
LIN {X 0,Y 432.306,Z 276.448,A -85,B 0,C 180,E1 -9477.077,E2 -9477.077} C_VEL
LIN {X 0,Y 432.339,Z 276.445,A -85,B 0,C 180,E1 -9480.259,E2 -9480.259} C_VEL
LIN {X 0,Y 432.334,Z 276.442,A -85,B 0,C 180,E1 -9483.551,E2 -9483.551} C_VEL
LIN {X 0,Y 432.332,Z 276.442,A -85,B 0,C 180,E1 -9485.817,E2 -9485.817} C_VEL
LIN {X 0,Y 432.321,Z 276.45,A -85,B 0,C 180,E1 -9489.344,E2 -9489.344} C_VEL
LIN {X 0,Y 432.317,Z 276.445,A -85,B 0,C 180,E1 -9491.797,E2 -9491.797} C_VEL
LIN {X 0,Y 432.326,Z 276.444,A -85,B 0,C 180,E1 -9494.347,E2 -9494.347} C_VEL
LIN {X 0,Y 432.312,Z 276.448,A -85,B 0,C 180,E1 -9497.015,E2 -9497.015} C_VEL
LIN {X 0,Y 432.325,Z 276.445,A -85,B 0,C 180,E1 -9499.82,E2 -9499.82} C_VEL
LIN {X 0,Y 432.297,Z 276.442,A -85,B 0,C 180,E1 -9503.021,E2 -9503.021} C_VEL
LIN {X 0,Y 432.35,Z 276.439,A -85,B 0,C 180,E1 -9505.996,E2 -9505.996} C_VEL
LIN {X 0,Y 432.336,Z 276.442,A -85,B 0,C 180,E1 -9509.489,E2 -9509.489} C_VEL
LIN {X 0,Y 432.379,Z 276.428,A -85,B 0,C 180,E1 -9512.928,E2 -9512.928} C_VEL
LIN {X 0,Y 432.356,Z 276.444,A -85,B 0,C 180,E1 -9516.023,E2 -9516.023} C_VEL
LIN {X 0,Y 432.337,Z 276.435,A -85,B 0,C 180,E1 -9519.046,E2 -9519.046} C_VEL
LIN {X 0,Y 432.364,Z 276.441,A -85,B 0,C 180,E1 -9522.011,E2 -9522.011} C_VEL
LIN {X 0,Y 432.381,Z 276.431,A -85,B 0,C 180,E1 -9524.926,E2 -9524.926} C_VEL
LIN {X 0,Y 432.447,Z 276.426,A -85,B 0,C 180,E1 -9527.803,E2 -9527.803} C_VEL
LIN {X 0,Y 432.479,Z 276.416,A -85,B 0,C 180,E1 -9531.59,E2 -9531.59} C_VEL
LIN {X 0,Y 432.582,Z 276.412,A -85,B 0,C 180,E1 -9534.406,E2 -9534.406} C_VEL
LIN {X 0,Y 432.589,Z 276.404,A -85,B 0,C 180,E1 -9538.138,E2 -9538.138} C_VEL
LIN {X 0,Y 432.719,Z 276.391,A -85,B 0,C 180,E1 -9540,E2 -9540} C_VEL
LIN {X 0,Y 432.579,Z 276.406,A -85,B 0,C 180,E1 -9542.794,E2 -9542.794} C_VEL
LIN {X 0,Y 432.573,Z 276.411,A -85,B 0,C 180,E1 -9545.594,E2 -9545.594} C_VEL
LIN {X 0,Y 432.47,Z 276.419,A -85,B 0,C 180,E1 -9548.41,E2 -9548.41} C_VEL
LIN {X 0,Y 432.447,Z 276.421,A -85,B 0,C 180,E1 -9552.197,E2 -9552.197} C_VEL
LIN {X 0,Y 432.419,Z 276.428,A -85,B 0,C 180,E1 -9556.039,E2 -9556.039} C_VEL
LIN {X 0,Y 432.376,Z 276.443,A -85,B 0,C 180,E1 -9559.486,E2 -9559.486} C_VEL
LIN {X 0,Y 432.308,Z 276.446,A -85,B 0,C 180,E1 -9562.965,E2 -9562.965} C_VEL
LIN {X 0,Y 432.355,Z 276.442,A -85,B 0,C 180,E1 -9566.033,E2 -9566.033} C_VEL
LIN {X 0,Y 432.343,Z 276.438,A -85,B 0,C 180,E1 -9569.188,E2 -9569.188} C_VEL
LIN {X 0,Y 432.317,Z 276.448,A -85,B 0,C 180,E1 -9572.294,E2 -9572.294} C_VEL
LIN {X 0,Y 432.333,Z 276.441,A -85,B 0,C 180,E1 -9574.678,E2 -9574.678} C_VEL
LIN {X 0,Y 432.343,Z 276.446,A -85,B 0,C 180,E1 -9578.149,E2 -9578.149} C_VEL
LIN {X 0,Y 432.37,Z 276.441,A -85,B 0,C 180,E1 -9581.61,E2 -9581.61} C_VEL
LIN {X 0,Y 432.432,Z 276.474,A -85,B 0,C 180,E1 -9582.729,E2 -9582.729} C_VEL
LIN {X 0,Y 432.94,Z 280.141,A -85,B 0,C 180,E1 -9583.623,E2 -9583.623} C_VEL
LIN {X 0,Y 432.563,Z 294.523,A -85,B 0,C 180,E1 -9586.971,E2 -9586.971} C_VEL
LIN {X 0,Y 432.54,Z 296.801,A -85,B 0,C 180,E1 -9587.499,E2 -9587.499} C_VEL
LIN {X 0,Y 435.229,Z 312.494,A -85,B 0,C 180,E1 -9587.884,E2 -9587.884} C_VEL
LIN {X 0,Y 434.625,Z 373.614,A -85,B 0,C 180,E1 -9588.935,E2 -9588.935} C_VEL
LIN {X 0,Y 434.423,Z 383.201,A -85,B 0,C 180,E1 -9589.223,E2 -9589.223} C_VEL
LIN {X 0,Y 434.189,Z 394.376,A -85,B 0,C 180,E1 -9589.727,E2 -9589.727} C_VEL
LIN {X 0,Y 433.737,Z 404.286,A -85,B 0,C 180,E1 -9590.358,E2 -9590.358} C_VEL
LIN {X 0,Y 433.313,Z 413.514,A -85,B 0,C 180,E1 -9591.126,E2 -9591.126} C_VEL
LIN {X 0,Y 432.9,Z 421.133,A -85,B 0,C 180,E1 -9591.91,E2 -9591.91} C_VEL
LIN {X 0,Y 432.515,Z 428.007,A -85,B 0,C 180,E1 -9592.77,E2 -9592.77} C_VEL
LIN {X 0,Y 432.236,Z 433.534,A -85,B 0,C 180,E1 -9593.597,E2 -9593.597} C_VEL
LIN {X 0,Y 431.934,Z 439.326,A -85,B 0,C 180,E1 -9594.642,E2 -9594.642} C_VEL
LIN {X 0,Y 431.704,Z 444.286,A -85,B 0,C 180,E1 -9595.747,E2 -9595.747} C_VEL
LIN {X 0,Y 431.456,Z 448.496,A -85,B 0,C 180,E1 -9596.93,E2 -9596.93} C_VEL
LIN {X 0,Y 431.402,Z 451.167,A -85,B 0,C 180,E1 -9597.902,E2 -9597.902} C_VEL
LIN {X 0,Y 431.304,Z 452.724,A -85,B 0,C 180,E1 -9598.573,E2 -9598.573} C_VEL
LIN {X 0,Y 431.192,Z 454.661,A -85,B 0,C 180,E1 -9599.752,E2 -9599.752} C_VEL
LIN {X 0,Y 431.073,Z 455.648,A -85,B 0,C 180,E1 -9600.719,E2 -9600.719} C_VEL
LIN {X 0,Y 431.049,Z 456.069,A -85,B 0,C 180,E1 -9601.783,E2 -9601.783} C_VEL
LIN {X 0,Y 431.029,Z 455.854,A -85,B 0,C 180,E1 -9602.837,E2 -9602.837} C_VEL
LIN {X 0,Y 431.095,Z 455.019,A -85,B 0,C 180,E1 -9603.886,E2 -9603.886} C_VEL
LIN {X 0,Y 431.184,Z 453.565,A -85,B 0,C 180,E1 -9604.927,E2 -9604.927} C_VEL
LIN {X 0,Y 431.375,Z 450.206,A -85,B 0,C 180,E1 -9606.475,E2 -9606.475} C_VEL
LIN {X 0,Y 431.619,Z 445.239,A -85,B 0,C 180,E1 -9608.007,E2 -9608.007} C_VEL
LIN {X 0,Y 431.837,Z 439.699,A -85,B 0,C 180,E1 -9609.27,E2 -9609.27} C_VEL
LIN {X 0,Y 432.158,Z 433.768,A -85,B 0,C 180,E1 -9610.349,E2 -9610.349} C_VEL
LIN {X 0,Y 432.5,Z 427.515,A -85,B 0,C 180,E1 -9611.281,E2 -9611.281} C_VEL
LIN {X 0,Y 432.886,Z 419.357,A -85,B 0,C 180,E1 -9612.278,E2 -9612.278} C_VEL
LIN {X 0,Y 433.405,Z 408.829,A -85,B 0,C 180,E1 -9613.275,E2 -9613.275} C_VEL
LIN {X 0,Y 433.766,Z 400.419,A -85,B 0,C 180,E1 -9613.892,E2 -9613.892} C_VEL
LIN {X 0,Y 434.069,Z 391.89,A -85,B 0,C 180,E1 -9614.385,E2 -9614.385} C_VEL
LIN {X 0,Y 434.281,Z 382.744,A -85,B 0,C 180,E1 -9614.784,E2 -9614.784} C_VEL
LIN {X 0,Y 434.496,Z 373.575,A -85,B 0,C 180,E1 -9615.058,E2 -9615.058} C_VEL
LIN {X 0,Y 433.834,Z 367.8,A -85,B 0,C 180,E1 -9615.204,E2 -9615.204} C_VEL
LIN {X 0,Y 428.482,Z 349.068,A -85,B 0,C 180,E1 -9615.689,E2 -9615.689} C_VEL
LIN {X 0,Y 427.885,Z 343.259,A -85,B 0,C 180,E1 -9615.805,E2 -9615.805} C_VEL
LIN {X 0,Y 427.947,Z 311.888,A -85,B 0,C 180,E1 -9616.346,E2 -9616.346} C_VEL
LIN {X 0,Y 425.465,Z 297.287,A -85,B 0,C 180,E1 -9616.709,E2 -9616.709} C_VEL
LIN {X 0,Y 425.913,Z 284.564,A -85,B 0,C 180,E1 -9620.023,E2 -9620.023} C_VEL
LIN {X 0,Y 425.614,Z 277.741,A -85,B 0,C 180,E1 -9621.848,E2 -9621.848} C_VEL
LIN {X 0,Y 425.543,Z 277.293,A -85,B 0,C 180,E1 -9621.978,E2 -9621.978} C_VEL
LIN {X 0,Y 425.552,Z 277.288,A -85,B 0,C 180,E1 -9624.313,E2 -9624.313} C_VEL
LIN {X 0,Y 425.575,Z 277.286,A -85,B 0,C 180,E1 -9628.107,E2 -9628.107} C_VEL
LIN {X 0,Y 425.704,Z 277.272,A -85,B 0,C 180,E1 -9630,E2 -9630} C_VEL
LIN {X 0,Y 425.548,Z 277.285,A -85,B 0,C 180,E1 -9632.84,E2 -9632.84} C_VEL
LIN {X 0,Y 425.542,Z 277.288,A -85,B 0,C 180,E1 -9635.687,E2 -9635.687} C_VEL
LIN {X 0,Y 425.438,Z 277.302,A -85,B 0,C 180,E1 -9638.55,E2 -9638.55} C_VEL
LIN {X 0,Y 425.413,Z 277.309,A -85,B 0,C 180,E1 -9642.401,E2 -9642.401} C_VEL
LIN {X 0,Y 425.389,Z 277.31,A -85,B 0,C 180,E1 -9646.311,E2 -9646.311} C_VEL
LIN {X 0,Y 425.328,Z 277.312,A -85,B 0,C 180,E1 -9649.635,E2 -9649.635} C_VEL
LIN {X 0,Y 425.288,Z 277.32,A -85,B 0,C 180,E1 -9652.338,E2 -9652.338} C_VEL
LIN {X 0,Y 425.291,Z 277.317,A -85,B 0,C 180,E1 -9655.445,E2 -9655.445} C_VEL
LIN {X 0,Y 425.33,Z 277.316,A -85,B 0,C 180,E1 -9658.631,E2 -9658.631} C_VEL
LIN {X 0,Y 425.261,Z 277.32,A -85,B 0,C 180,E1 -9661.926,E2 -9661.926} C_VEL
LIN {X 0,Y 425.294,Z 277.322,A -85,B 0,C 180,E1 -9665.335,E2 -9665.335} C_VEL
LIN {X 0,Y 425.293,Z 277.321,A -85,B 0,C 180,E1 -9669.042,E2 -9669.042} C_VEL
LIN {X 0,Y 425.27,Z 277.319,A -85,B 0,C 180,E1 -9672.652,E2 -9672.652} C_VEL
LIN {X 0,Y 425.313,Z 277.316,A -85,B 0,C 180,E1 -9676.051,E2 -9676.051} C_VEL
LIN {X 0,Y 425.303,Z 277.315,A -85,B 0,C 180,E1 -9678.625,E2 -9678.625} C_VEL
LIN {X 0,Y 425.315,Z 277.315,A -85,B 0,C 180,E1 -9681.103,E2 -9681.103} C_VEL
LIN {X 0,Y 425.293,Z 277.316,A -85,B 0,C 180,E1 -9684.663,E2 -9684.663} C_VEL
LIN {X 0,Y 425.258,Z 277.327,A -85,B 0,C 180,E1 -9688.072,E2 -9688.072} C_VEL
LIN {X 0,Y 425.329,Z 277.312,A -85,B 0,C 180,E1 -9691.368,E2 -9691.368} C_VEL
LIN {X 0,Y 425.286,Z 277.321,A -85,B 0,C 180,E1 -9694.554,E2 -9694.554} C_VEL
LIN {X 0,Y 425.277,Z 277.319,A -85,B 0,C 180,E1 -9697.661,E2 -9697.661} C_VEL
LIN {X 0,Y 425.351,Z 277.313,A -85,B 0,C 180,E1 -9700.703,E2 -9700.703} C_VEL
LIN {X 0,Y 425.377,Z 277.306,A -85,B 0,C 180,E1 -9703.688,E2 -9703.688} C_VEL
LIN {X 0,Y 425.4,Z 277.303,A -85,B 0,C 180,E1 -9707.598,E2 -9707.598} C_VEL
LIN {X 0,Y 425.43,Z 277.3,A -85,B 0,C 180,E1 -9711.45,E2 -9711.45} C_VEL
LIN {X 0,Y 425.537,Z 277.287,A -85,B 0,C 180,E1 -9714.313,E2 -9714.313} C_VEL
LIN {X 0,Y 425.563,Z 277.282,A -85,B 0,C 180,E1 -9718.107,E2 -9718.107} C_VEL
LIN {X 0,Y 425.689,Z 277.267,A -85,B 0,C 180,E1 -9720,E2 -9720} C_VEL
LIN {X 0,Y 425.534,Z 277.29,A -85,B 0,C 180,E1 -9722.84,E2 -9722.84} C_VEL
LIN {X 0,Y 425.515,Z 277.289,A -85,B 0,C 180,E1 -9726.639,E2 -9726.639} C_VEL
LIN {X 0,Y 425.392,Z 277.311,A -85,B 0,C 180,E1 -9729.509,E2 -9729.509} C_VEL
LIN {X 0,Y 425.392,Z 277.305,A -85,B 0,C 180,E1 -9732.91,E2 -9732.91} C_VEL
LIN {X 0,Y 425.35,Z 277.309,A -85,B 0,C 180,E1 -9736.605,E2 -9736.605} C_VEL
LIN {X 0,Y 425.317,Z 277.319,A -85,B 0,C 180,E1 -9739.636,E2 -9739.636} C_VEL
LIN {X 0,Y 425.277,Z 277.321,A -85,B 0,C 180,E1 -9742.339,E2 -9742.339} C_VEL
LIN {X 0,Y 425.285,Z 277.319,A -85,B 0,C 180,E1 -9745.446,E2 -9745.446} C_VEL
LIN {X 0,Y 425.32,Z 277.315,A -85,B 0,C 180,E1 -9748.633,E2 -9748.633} C_VEL
LIN {X 0,Y 425.255,Z 277.325,A -85,B 0,C 180,E1 -9751.928,E2 -9751.928} C_VEL
LIN {X 0,Y 425.291,Z 277.316,A -85,B 0,C 180,E1 -9755.337,E2 -9755.337} C_VEL
LIN {X 0,Y 425.284,Z 277.32,A -85,B 0,C 180,E1 -9758.9,E2 -9758.9} C_VEL
LIN {X 0,Y 425.282,Z 277.319,A -85,B 0,C 180,E1 -9761.959,E2 -9761.959} C_VEL
LIN {X 0,Y 425.278,Z 277.32,A -85,B 0,C 180,E1 -9765.284,E2 -9765.284} C_VEL
LIN {X 0,Y 425.261,Z 277.326,A -85,B 0,C 180,E1 -9768.621,E2 -9768.621} C_VEL
LIN {X 0,Y 425.291,Z 277.322,A -85,B 0,C 180,E1 -9771.102,E2 -9771.102} C_VEL
LIN {X 0,Y 425.293,Z 277.319,A -85,B 0,C 180,E1 -9774.665,E2 -9774.665} C_VEL
LIN {X 0,Y 425.259,Z 277.32,A -85,B 0,C 180,E1 -9778.074,E2 -9778.074} C_VEL
LIN {X 0,Y 425.307,Z 277.322,A -85,B 0,C 180,E1 -9781.367,E2 -9781.367} C_VEL
LIN {X 0,Y 425.266,Z 277.323,A -85,B 0,C 180,E1 -9784.554,E2 -9784.554} C_VEL
LIN {X 0,Y 425.361,Z 277.427,A -85,B 0,C 180,E1 -9785.564,E2 -9785.564} C_VEL
LIN {X 0,Y 426.827,Z 286.351,A -85,B 0,C 180,E1 -9787.747,E2 -9787.747} C_VEL
LIN {X 0,Y 426.574,Z 293.949,A -85,B 0,C 180,E1 -9789.507,E2 -9789.507} C_VEL
LIN {X 0,Y 425.729,Z 310.295,A -85,B 0,C 180,E1 -9793.23,E2 -9793.23} C_VEL
LIN {X 0,Y 425.284,Z 319.733,A -85,B 0,C 180,E1 -9795.343,E2 -9795.343} C_VEL
LIN {X 0,Y 427.99,Z 341.161,A -85,B 0,C 180,E1 -9795.803,E2 -9795.803} C_VEL
LIN {X 0,Y 427.485,Z 397.217,A -85,B 0,C 180,E1 -9796.784,E2 -9796.784} C_VEL
LIN {X 0,Y 427.138,Z 407.6,A -85,B 0,C 180,E1 -9797.106,E2 -9797.106} C_VEL
LIN {X 0,Y 426.734,Z 418.786,A -85,B 0,C 180,E1 -9797.638,E2 -9797.638} C_VEL
LIN {X 0,Y 426.261,Z 429.292,A -85,B 0,C 180,E1 -9798.348,E2 -9798.348} C_VEL
LIN {X 0,Y 425.877,Z 437.554,A -85,B 0,C 180,E1 -9799.061,E2 -9799.061} C_VEL
LIN {X 0,Y 425.477,Z 445.388,A -85,B 0,C 180,E1 -9799.892,E2 -9799.892} C_VEL
LIN {X 0,Y 425.132,Z 451.863,A -85,B 0,C 180,E1 -9800.725,E2 -9800.725} C_VEL
LIN {X 0,Y 424.757,Z 458.028,A -85,B 0,C 180,E1 -9801.676,E2 -9801.676} C_VEL
LIN {X 0,Y 424.543,Z 464.327,A -85,B 0,C 180,E1 -9802.868,E2 -9802.868} C_VEL
LIN {X 0,Y 424.283,Z 470.166,A -85,B 0,C 180,E1 -9804.296,E2 -9804.296} C_VEL
LIN {X 0,Y 424.234,Z 473.203,A -85,B 0,C 180,E1 -9805.249,E2 -9805.249} C_VEL
LIN {X 0,Y 424.126,Z 475.557,A -85,B 0,C 180,E1 -9806.2,E2 -9806.2} C_VEL
LIN {X 0,Y 424.143,Z 477.356,A -85,B 0,C 180,E1 -9807.151,E2 -9807.151} C_VEL
LIN {X 0,Y 424.129,Z 478.649,A -85,B 0,C 180,E1 -9808.101,E2 -9808.101} C_VEL
LIN {X 0,Y 424.086,Z 479.462,A -85,B 0,C 180,E1 -9809.05,E2 -9809.05} C_VEL
LIN {X 0,Y 424.083,Z 479.765,A -85,B 0,C 180,E1 -9810,E2 -9810} C_VEL
LIN {X 0,Y 424.086,Z 479.478,A -85,B 0,C 180,E1 -9810.95,E2 -9810.95} C_VEL
LIN {X 0,Y 424.129,Z 478.717,A -85,B 0,C 180,E1 -9811.899,E2 -9811.899} C_VEL
LIN {X 0,Y 424.142,Z 477.477,A -85,B 0,C 180,E1 -9812.849,E2 -9812.849} C_VEL
LIN {X 0,Y 424.161,Z 474.572,A -85,B 0,C 180,E1 -9814.276,E2 -9814.276} C_VEL
LIN {X 0,Y 424.276,Z 471.935,A -85,B 0,C 180,E1 -9815.227,E2 -9815.227} C_VEL
LIN {X 0,Y 424.405,Z 467.39,A -85,B 0,C 180,E1 -9816.497,E2 -9816.497} C_VEL
LIN {X 0,Y 424.58,Z 462.355,A -85,B 0,C 180,E1 -9817.609,E2 -9817.609} C_VEL
LIN {X 0,Y 424.849,Z 457.097,A -85,B 0,C 180,E1 -9818.562,E2 -9818.562} C_VEL
LIN {X 0,Y 425.259,Z 450.775,A -85,B 0,C 180,E1 -9819.512,E2 -9819.512} C_VEL
LIN {X 0,Y 425.75,Z 442.063,A -85,B 0,C 180,E1 -9820.582,E2 -9820.582} C_VEL
LIN {X 0,Y 426.254,Z 432.023,A -85,B 0,C 180,E1 -9821.532,E2 -9821.532} C_VEL
LIN {X 0,Y 426.638,Z 424.131,A -85,B 0,C 180,E1 -9822.124,E2 -9822.124} C_VEL
LIN {X 0,Y 427.016,Z 415.088,A -85,B 0,C 180,E1 -9822.656,E2 -9822.656} C_VEL
LIN {X 0,Y 427.378,Z 405.64,A -85,B 0,C 180,E1 -9823.068,E2 -9823.068} C_VEL
LIN {X 0,Y 427.67,Z 396.721,A -85,B 0,C 180,E1 -9823.334,E2 -9823.334} C_VEL
LIN {X 0,Y 428.1,Z 339.547,A -85,B 0,C 180,E1 -9824.341,E2 -9824.341} C_VEL
LIN {X 0,Y 425.301,Z 319.072,A -85,B 0,C 180,E1 -9824.825,E2 -9824.825} C_VEL
LIN {X 0,Y 426.042,Z 303.509,A -85,B 0,C 180,E1 -9828.265,E2 -9828.265} C_VEL
LIN {X 0,Y 426.786,Z 287.962,A -85,B 0,C 180,E1 -9831.747,E2 -9831.747} C_VEL
LIN {X 0,Y 426.544,Z 283.946,A -85,B 0,C 180,E1 -9832.678,E2 -9832.678} C_VEL
LIN {X 0,Y 425.336,Z 277.32,A -85,B 0,C 180,E1 -9834.301,E2 -9834.301} C_VEL
LIN {X 0,Y 425.255,Z 277.325,A -85,B 0,C 180,E1 -9837.563,E2 -9837.563} C_VEL
LIN {X 0,Y 425.286,Z 277.324,A -85,B 0,C 180,E1 -9840.76,E2 -9840.76} C_VEL
LIN {X 0,Y 425.304,Z 277.318,A -85,B 0,C 180,E1 -9844.287,E2 -9844.287} C_VEL
LIN {X 0,Y 425.273,Z 277.325,A -85,B 0,C 180,E1 -9847.694,E2 -9847.694} C_VEL
LIN {X 0,Y 425.27,Z 277.325,A -85,B 0,C 180,E1 -9850.519,E2 -9850.519} C_VEL
LIN {X 0,Y 425.253,Z 277.326,A -85,B 0,C 180,E1 -9853.955,E2 -9853.955} C_VEL
LIN {X 0,Y 425.267,Z 277.329,A -85,B 0,C 180,E1 -9857.346,E2 -9857.346} C_VEL
LIN {X 0,Y 425.277,Z 277.323,A -85,B 0,C 180,E1 -9859.872,E2 -9859.872} C_VEL
LIN {X 0,Y 425.268,Z 277.316,A -85,B 0,C 180,E1 -9862.488,E2 -9862.488} C_VEL
LIN {X 0,Y 425.298,Z 277.32,A -85,B 0,C 180,E1 -9865.817,E2 -9865.817} C_VEL
LIN {X 0,Y 425.28,Z 277.318,A -85,B 0,C 180,E1 -9869.238,E2 -9869.238} C_VEL
LIN {X 0,Y 425.337,Z 277.307,A -85,B 0,C 180,E1 -9872.442,E2 -9872.442} C_VEL
LIN {X 0,Y 425.336,Z 277.314,A -85,B 0,C 180,E1 -9875.601,E2 -9875.601} C_VEL
LIN {X 0,Y 425.281,Z 277.316,A -85,B 0,C 180,E1 -9878.681,E2 -9878.681} C_VEL
LIN {X 0,Y 425.32,Z 277.315,A -85,B 0,C 180,E1 -9881.702,E2 -9881.702} C_VEL
LIN {X 0,Y 425.335,Z 277.31,A -85,B 0,C 180,E1 -9884.67,E2 -9884.67} C_VEL
LIN {X 0,Y 425.4,Z 277.304,A -85,B 0,C 180,E1 -9887.598,E2 -9887.598} C_VEL
LIN {X 0,Y 425.43,Z 277.295,A -85,B 0,C 180,E1 -9891.45,E2 -9891.45} C_VEL
LIN {X 0,Y 425.539,Z 277.288,A -85,B 0,C 180,E1 -9894.313,E2 -9894.313} C_VEL
LIN {X 0,Y 425.559,Z 277.28,A -85,B 0,C 180,E1 -9898.107,E2 -9898.107} C_VEL
LIN {X 0,Y 425.689,Z 277.266,A -85,B 0,C 180,E1 -9900,E2 -9900} C_VEL
LIN {X 0,Y 425.533,Z 277.284,A -85,B 0,C 180,E1 -9902.84,E2 -9902.84} C_VEL
LIN {X 0,Y 425.485,Z 277.293,A -85,B 0,C 180,E1 -9906.511,E2 -9906.511} C_VEL
LIN {X 0,Y 425.388,Z 277.311,A -85,B 0,C 180,E1 -9909.51,E2 -9909.51} C_VEL
LIN {X 0,Y 425.381,Z 277.303,A -85,B 0,C 180,E1 -9912.904,E2 -9912.904} C_VEL
LIN {X 0,Y 425.35,Z 277.307,A -85,B 0,C 180,E1 -9916.605,E2 -9916.605} C_VEL
LIN {X 0,Y 425.317,Z 277.32,A -85,B 0,C 180,E1 -9919.636,E2 -9919.636} C_VEL
LIN {X 0,Y 425.296,Z 277.322,A -85,B 0,C 180,E1 -9923.366,E2 -9923.366} C_VEL
LIN {X 0,Y 425.339,Z 277.311,A -85,B 0,C 180,E1 -9926.845,E2 -9926.845} C_VEL
LIN {X 0,Y 425.309,Z 277.319,A -85,B 0,C 180,E1 -9929.718,E2 -9929.718} C_VEL
LIN {X 0,Y 425.274,Z 277.321,A -85,B 0,C 180,E1 -9933.049,E2 -9933.049} C_VEL
LIN {X 0,Y 425.277,Z 277.322,A -85,B 0,C 180,E1 -9935.93,E2 -9935.93} C_VEL
LIN {X 0,Y 425.303,Z 277.319,A -85,B 0,C 180,E1 -9939.046,E2 -9939.046} C_VEL
LIN {X 0,Y 425.4,Z 277.435,A -85,B 0,C 180,E1 -9942.585,E2 -9942.585} C_VEL
LIN {X 0,Y 425.949,Z 282.673,A -85,B 0,C 180,E1 -9943.867,E2 -9943.867} C_VEL
LIN {X 0,Y 425.56,Z 297.034,A -85,B 0,C 180,E1 -9947.255,E2 -9947.255} C_VEL
LIN {X 0,Y 428.387,Z 313.14,A -85,B 0,C 180,E1 -9947.648,E2 -9947.648} C_VEL
LIN {X 0,Y 427.734,Z 374.185,A -85,B 0,C 180,E1 -9948.717,E2 -9948.717} C_VEL
LIN {X 0,Y 427.512,Z 385.152,A -85,B 0,C 180,E1 -9949.065,E2 -9949.065} C_VEL
LIN {X 0,Y 427.181,Z 396.454,A -85,B 0,C 180,E1 -9949.626,E2 -9949.626} C_VEL
LIN {X 0,Y 426.753,Z 405.69,A -85,B 0,C 180,E1 -9950.251,E2 -9950.251} C_VEL
LIN {X 0,Y 426.329,Z 414.203,A -85,B 0,C 180,E1 -9950.983,E2 -9950.983} C_VEL
LIN {X 0,Y 425.908,Z 421.674,A -85,B 0,C 180,E1 -9951.773,E2 -9951.773} C_VEL
LIN {X 0,Y 425.496,Z 428.711,A -85,B 0,C 180,E1 -9952.678,E2 -9952.678} C_VEL
LIN {X 0,Y 425.104,Z 436.069,A -85,B 0,C 180,E1 -9953.843,E2 -9953.843} C_VEL
LIN {X 0,Y 424.728,Z 442.71,A -85,B 0,C 180,E1 -9955.19,E2 -9955.19} C_VEL
LIN {X 0,Y 424.444,Z 447.181,A -85,B 0,C 180,E1 -9956.359,E2 -9956.359} C_VEL
LIN {X 0,Y 424.338,Z 450.916,A -85,B 0,C 180,E1 -9957.637,E2 -9957.637} C_VEL
LIN {X 0,Y 424.149,Z 453.916,A -85,B 0,C 180,E1 -9959.093,E2 -9959.093} C_VEL
LIN {X 0,Y 424.036,Z 455.342,A -85,B 0,C 180,E1 -9960.185,E2 -9960.185} C_VEL
LIN {X 0,Y 423.945,Z 456.17,A -85,B 0,C 180,E1 -9961.476,E2 -9961.476} C_VEL
LIN {X 0,Y 423.926,Z 456.223,A -85,B 0,C 180,E1 -9962.343,E2 -9962.343} C_VEL
LIN {X 0,Y 423.984,Z 455.607,A -85,B 0,C 180,E1 -9963.523,E2 -9963.523} C_VEL
LIN {X 0,Y 424.038,Z 454.589,A -85,B 0,C 180,E1 -9964.475,E2 -9964.475} C_VEL
LIN {X 0,Y 424.207,Z 452.496,A -85,B 0,C 180,E1 -9965.673,E2 -9965.673} C_VEL
LIN {X 0,Y 424.398,Z 448.789,A -85,B 0,C 180,E1 -9967.099,E2 -9967.099} C_VEL
LIN {X 0,Y 424.587,Z 444.552,A -85,B 0,C 180,E1 -9968.315,E2 -9968.315} C_VEL
LIN {X 0,Y 424.815,Z 439.699,A -85,B 0,C 180,E1 -9969.418,E2 -9969.418} C_VEL
LIN {X 0,Y 425.108,Z 434.13,A -85,B 0,C 180,E1 -9970.448,E2 -9970.448} C_VEL
LIN {X 0,Y 425.396,Z 429.264,A -85,B 0,C 180,E1 -9971.207,E2 -9971.207} C_VEL
LIN {X 0,Y 425.719,Z 422.5,A -85,B 0,C 180,E1 -9972.094,E2 -9972.094} C_VEL
LIN {X 0,Y 426.168,Z 414.716,A -85,B 0,C 180,E1 -9972.93,E2 -9972.93} C_VEL
LIN {X 0,Y 426.563,Z 406.634,A -85,B 0,C 180,E1 -9973.637,E2 -9973.637} C_VEL
LIN {X 0,Y 426.977,Z 397.017,A -85,B 0,C 180,E1 -9974.303,E2 -9974.303} C_VEL
LIN {X 0,Y 427.301,Z 385.359,A -85,B 0,C 180,E1 -9974.895,E2 -9974.895} C_VEL
LIN {X 0,Y 427.578,Z 374.619,A -85,B 0,C 180,E1 -9975.241,E2 -9975.241} C_VEL
LIN {X 0,Y 427.831,Z 346.997,A -85,B 0,C 180,E1 -9975.742,E2 -9975.742} C_VEL
LIN {X 0,Y 427.885,Z 343.259,A -85,B 0,C 180,E1 -9975.805,E2 -9975.805} C_VEL
LIN {X 0,Y 427.097,Z 335.536,A -85,B 0,C 180,E1 -9975.964,E2 -9975.964} C_VEL
LIN {X 0,Y 421.091,Z 312.94,A -85,B 0,C 180,E1 -9976.555,E2 -9976.555} C_VEL
LIN {X 0,Y 418.464,Z 297.524,A -85,B 0,C 180,E1 -9976.931,E2 -9976.931} C_VEL
LIN {X 0,Y 418.933,Z 284.623,A -85,B 0,C 180,E1 -9980.343,E2 -9980.343} C_VEL
LIN {X 0,Y 418.521,Z 278.322,A -85,B 0,C 180,E1 -9982.062,E2 -9982.062} C_VEL
LIN {X 0,Y 418.511,Z 278.166,A -85,B 0,C 180,E1 -9984.217,E2 -9984.217} C_VEL
LIN {X 0,Y 418.544,Z 278.162,A -85,B 0,C 180,E1 -9988.076,E2 -9988.076} C_VEL
LIN {X 0,Y 418.673,Z 278.148,A -85,B 0,C 180,E1 -9990,E2 -9990} C_VEL
LIN {X 0,Y 418.503,Z 278.162,A -85,B 0,C 180,E1 -9992.888,E2 -9992.888} C_VEL
LIN {X 0,Y 418.5,Z 278.166,A -85,B 0,C 180,E1 -9995.783,E2 -9995.783} C_VEL
LIN {X 0,Y 418.398,Z 278.177,A -85,B 0,C 180,E1 -9998.695,E2 -9998.695} C_VEL
